   1:L PR[91] R[100]mm/sec CNT100;
   1:  PR[GP1:91,1] = PR[GP1:90,1] + -46.365;
   1:  PR[GP1:91,2] = PR[GP1:90,2] + -31.306;
   1:L PR[91] R[100]mm/sec CNT100;
   1:  PR[GP1:91,1] = PR[GP1:90,1] + -43.823;
   1:  PR[GP1:91,2] = PR[GP1:90,2] + -32.890;
   1:L PR[91] R[100]mm/sec CNT100;
   1:  PR[GP1:91,1] = PR[GP1:90,1] + -41.333;
   1:  PR[GP1:91,2] = PR[GP1:90,2] + -33.889;
   1:L PR[91] R[100]mm/sec CNT100;
   1:  PR[GP1:91,1] = PR[GP1:90,1] + -32.971;
   1:  PR[GP1:91,2] = PR[GP1:90,2] + -36.840;
   1:L PR[91] R[100]mm/sec CNT100;
   1:  PR[GP1:91,1] = PR[GP1:90,1] + -30.718;
   1:  PR[GP1:91,2] = PR[GP1:90,2] + -37.326;
   1:L PR[91] R[100]mm/sec CNT100;
   1:  PR[GP1:91,1] = PR[GP1:90,1] + -28.669;
   1:  PR[GP1:91,2] = PR[GP1:90,2] + -37.405;
   1:L PR[91] R[100]mm/sec CNT100;
   1:  PR[GP1:91,1] = PR[GP1:90,1] + -18.411;
   1:  PR[GP1:91,2] = PR[GP1:90,2] + -37.437;
   1:L PR[91] R[100]mm/sec CNT100;
   1:  PR[GP1:91,1] = PR[GP1:90,1] + -16.830;
   1:  PR[GP1:91,2] = PR[GP1:90,2] + -37.231;
   1:L PR[91] R[100]mm/sec CNT100;
   1:  PR[GP1:91,1] = PR[GP1:90,1] + -15.463;
   1:  PR[GP1:91,2] = PR[GP1:90,2] + -36.795;
   1:L PR[91] R[100]mm/sec CNT100;
   1:  PR[GP1:91,1] = PR[GP1:90,1] + -4.794;
   1:  PR[GP1:91,2] = PR[GP1:90,2] + -33.088;
   1:L PR[91] R[100]mm/sec CNT100;
   1:  PR[GP1:91,1] = PR[GP1:90,1] + -3.959;
   1:  PR[GP1:91,2] = PR[GP1:90,2] + -32.651;
   1:L PR[91] R[100]mm/sec CNT100;
   1:  PR[GP1:91,1] = PR[GP1:90,1] + -2.575;
   1:  PR[GP1:91,2] = PR[GP1:90,2] + -31.645;
   1:L PR[91] R[100]mm/sec CNT100;
   1:  PR[GP1:91,1] = PR[GP1:90,1] + -0.246;
   1:  PR[GP1:91,2] = PR[GP1:90,2] + -31.552;
   1:L PR[91] R[100]mm/sec CNT100;
   1:  PR[GP1:91,1] = PR[GP1:90,1] + 1.907;
   1:  PR[GP1:91,2] = PR[GP1:90,2] + -31.093;
   1:L PR[91] R[100]mm/sec CNT100;
   1:  PR[GP1:91,1] = PR[GP1:90,1] + 2.367;
   1:  PR[GP1:91,2] = PR[GP1:90,2] + -31.464;
   1:L PR[91] R[100]mm/sec CNT100;
   1:  PR[GP1:91,1] = PR[GP1:90,1] + 2.888;
   1:  PR[GP1:91,2] = PR[GP1:90,2] + -31.723;
   1:L PR[91] R[100]mm/sec CNT100;
   1:  PR[GP1:91,1] = PR[GP1:90,1] + 4.168;
   1:  PR[GP1:91,2] = PR[GP1:90,2] + -32.653;
   1:L PR[91] R[100]mm/sec CNT100;
   1:  PR[GP1:91,1] = PR[GP1:90,1] + 4.991;
   1:  PR[GP1:91,2] = PR[GP1:90,2] + -33.083;
   1:L PR[91] R[100]mm/sec CNT100;
   1:  PR[GP1:91,1] = PR[GP1:90,1] + 6.059;
   1:  PR[GP1:91,2] = PR[GP1:90,2] + -33.426;
   1:L PR[91] R[100]mm/sec CNT100;
   1:  PR[GP1:91,1] = PR[GP1:90,1] + 17.047;
   1:  PR[GP1:91,2] = PR[GP1:90,2] + -37.230;
   1:L PR[91] R[100]mm/sec CNT100;
   1:  PR[GP1:91,1] = PR[GP1:90,1] + 18.609;
   1:  PR[GP1:91,2] = PR[GP1:90,2] + -37.435;
   1:L PR[91] R[100]mm/sec CNT100;
   1:  PR[GP1:91,1] = PR[GP1:90,1] + 20.489;
   1:  PR[GP1:91,2] = PR[GP1:90,2] + -37.372;
   1:L PR[91] R[100]mm/sec CNT100;
   1:  PR[GP1:91,1] = PR[GP1:90,1] + 30.926;
   1:  PR[GP1:91,2] = PR[GP1:90,2] + -37.326;
   1:L PR[91] R[100]mm/sec CNT100;
   1:  PR[GP1:91,1] = PR[GP1:90,1] + 33.154;
   1:  PR[GP1:91,2] = PR[GP1:90,2] + -36.847;
   1:L PR[91] R[100]mm/sec CNT100;
   1:  PR[GP1:91,1] = PR[GP1:90,1] + 35.646;
   1:  PR[GP1:91,2] = PR[GP1:90,2] + -35.865;
   1:L PR[91] R[100]mm/sec CNT100;
   1:  PR[GP1:91,1] = PR[GP1:90,1] + 44.032;
   1:  PR[GP1:91,2] = PR[GP1:90,2] + -32.893;
   1:L PR[91] R[100]mm/sec CNT100;
   1:  PR[GP1:91,1] = PR[GP1:90,1] + 46.535;
   1:  PR[GP1:91,2] = PR[GP1:90,2] + -31.341;
   1:L PR[91] R[100]mm/sec CNT100;
   1:  PR[GP1:91,1] = PR[GP1:90,1] + 48.999;
   1:  PR[GP1:91,2] = PR[GP1:90,2] + -29.159;
   1:L PR[91] R[100]mm/sec CNT100;
   1:  PR[GP1:91,1] = PR[GP1:90,1] + 54.738;
   1:  PR[GP1:91,2] = PR[GP1:90,2] + -24.513;
   1:L PR[91] R[100]mm/sec CNT100;
   1:  PR[GP1:91,1] = PR[GP1:90,1] + 56.858;
   1:  PR[GP1:91,2] = PR[GP1:90,2] + -21.761;
   1:L PR[91] R[100]mm/sec CNT100;
   1:  PR[GP1:91,1] = PR[GP1:90,1] + 58.644;
   1:  PR[GP1:91,2] = PR[GP1:90,2] + -18.336;
   1:L PR[91] R[100]mm/sec CNT100;
   1:  PR[GP1:91,1] = PR[GP1:90,1] + 61.851;
   1:  PR[GP1:91,2] = PR[GP1:90,2] + -12.992;
   1:L PR[91] R[100]mm/sec CNT100;
   1:  PR[GP1:91,1] = PR[GP1:90,1] + 62.889;
   1:  PR[GP1:91,2] = PR[GP1:90,2] + -9.519;
   1:L PR[91] R[100]mm/sec CNT100;
   1:  PR[GP1:91,1] = PR[GP1:90,1] + 63.252;
   1:  PR[GP1:91,2] = PR[GP1:90,2] + -5.632;
   1:L PR[91] R[100]mm/sec CNT100;
   1:  PR[GP1:91,1] = PR[GP1:90,1] + 64.281;
   1:  PR[GP1:91,2] = PR[GP1:90,2] + -0.045;
   1:L PR[91] R[100]mm/sec CNT100;
   1:  PR[GP1:91,1] = PR[GP1:90,1] + 63.927;
   1:  PR[GP1:91,2] = PR[GP1:90,2] + 3.792;
   1:L PR[91] R[100]mm/sec CNT100;
   1:  PR[GP1:91,1] = PR[GP1:90,1] + 62.897;
   1:  PR[GP1:91,2] = PR[GP1:90,2] + 9.347;
   1:L PR[91] R[100]mm/sec CNT100;
   1:  PR[GP1:91,1] = PR[GP1:90,1] + 61.846;
   1:  PR[GP1:91,2] = PR[GP1:90,2] + 12.865;
   1:L PR[91] R[100]mm/sec CNT100;
   1:  PR[GP1:91,1] = PR[GP1:90,1] + 60.137;
   1:  PR[GP1:91,2] = PR[GP1:90,2] + 16.178;
   1:L PR[91] R[100]mm/sec CNT100;
   1:  PR[GP1:91,1] = PR[GP1:90,1] + 56.873;
   1:  PR[GP1:91,2] = PR[GP1:90,2] + 21.599;
   1:L PR[91] R[100]mm/sec CNT100;
   1:  PR[GP1:91,1] = PR[GP1:90,1] + 54.732;
   1:  PR[GP1:91,2] = PR[GP1:90,2] + 24.378;
   1:L PR[91] R[100]mm/sec CNT100;
   1:  PR[GP1:91,1] = PR[GP1:90,1] + 52.362;
   1:  PR[GP1:91,2] = PR[GP1:90,2] + 26.497;
   1:L PR[91] R[100]mm/sec CNT100;
   1:  PR[GP1:91,1] = PR[GP1:90,1] + 46.553;
   1:  PR[GP1:91,2] = PR[GP1:90,2] + 31.186;
   1:L PR[91] R[100]mm/sec CNT100;
   1:  PR[GP1:91,1] = PR[GP1:90,1] + 44.028;
   1:  PR[GP1:91,2] = PR[GP1:90,2] + 32.752;
   1:L PR[91] R[100]mm/sec CNT100;
   1:  PR[GP1:91,1] = PR[GP1:90,1] + 41.535;
   1:  PR[GP1:91,2] = PR[GP1:90,2] + 33.747;
   1:L PR[91] R[100]mm/sec CNT100;
   1:  PR[GP1:91,1] = PR[GP1:90,1] + 33.176;
   1:  PR[GP1:91,2] = PR[GP1:90,2] + 36.698;
   1:L PR[91] R[100]mm/sec CNT100;
   1:  PR[GP1:91,1] = PR[GP1:90,1] + 30.927;
   1:  PR[GP1:91,2] = PR[GP1:90,2] + 37.182;
   1:L PR[91] R[100]mm/sec CNT100;
   1:  PR[GP1:91,1] = PR[GP1:90,1] + 28.888;
   1:  PR[GP1:91,2] = PR[GP1:90,2] + 37.259;
   1:L PR[91] R[100]mm/sec CNT100;
   1:  PR[GP1:91,1] = PR[GP1:90,1] + 18.635;
   1:  PR[GP1:91,2] = PR[GP1:90,2] + 37.295;
   1:L PR[91] R[100]mm/sec CNT100;
   1:  PR[GP1:91,1] = PR[GP1:90,1] + 17.056;
   1:  PR[GP1:91,2] = PR[GP1:90,2] + 37.088;
   1:L PR[91] R[100]mm/sec CNT100;
   1:  PR[GP1:91,1] = PR[GP1:90,1] + 15.687;
   1:  PR[GP1:91,2] = PR[GP1:90,2] + 36.652;
   1:L PR[91] R[100]mm/sec CNT100;
   1:  PR[GP1:91,1] = PR[GP1:90,1] + 5.015;
   1:  PR[GP1:91,2] = PR[GP1:90,2] + 32.952;
   1:L PR[91] R[100]mm/sec CNT100;
   1:  PR[GP1:91,1] = PR[GP1:90,1] + 4.175;
   1:  PR[GP1:91,2] = PR[GP1:90,2] + 32.514;
   1:L PR[91] R[100]mm/sec CNT100;
   1:  PR[GP1:91,1] = PR[GP1:90,1] + 3.190;
   1:  PR[GP1:91,2] = PR[GP1:90,2] + 31.818;
   1:L PR[91] R[100]mm/sec CNT100;
   1:  PR[GP1:91,1] = PR[GP1:90,1] + 3.196;
   1:  PR[GP1:91,2] = PR[GP1:90,2] + 31.710;
   1:L PR[91] R[100]mm/sec CNT100;
   1:  PR[GP1:91,1] = PR[GP1:90,1] + 1.880;
   1:  PR[GP1:91,2] = PR[GP1:90,2] + 30.978;
   1:L PR[91] R[100]mm/sec CNT100;
   1:  ! -- Layer/Ebene 107 -- !;
   1:  PR[91] = PR[90];
   1:  PR[GP1:91,1] = PR[GP1:90,1] + -1.357;
   1:  PR[GP1:91,2] = PR[GP1:90,2] + 31.489;
   1:  PR[GP1:91,3] = PR[GP1:90,3] + 65.575;
   1:L PR[91] R[100]mm/sec CNT100;
   1:  PR[GP1:91,1] = PR[GP1:90,1] + -2.590;
   1:  PR[GP1:91,2] = PR[GP1:90,2] + 31.776;
   1:L PR[91] R[100]mm/sec CNT100;
   1:  PR[GP1:91,1] = PR[GP1:90,1] + -3.756;
   1:  PR[GP1:91,2] = PR[GP1:90,2] + 32.599;
   1:L PR[91] R[100]mm/sec CNT100;
   1:  PR[GP1:91,1] = PR[GP1:90,1] + -4.464;
   1:  PR[GP1:91,2] = PR[GP1:90,2] + 32.970;
   1:L PR[91] R[100]mm/sec CNT100;
   1:  PR[GP1:91,1] = PR[GP1:90,1] + -5.379;
   1:  PR[GP1:91,2] = PR[GP1:90,2] + 33.264;
   1:L PR[91] R[100]mm/sec CNT100;
   1:  PR[GP1:91,1] = PR[GP1:90,1] + -16.656;
   1:  PR[GP1:91,2] = PR[GP1:90,2] + 37.163;
   1:L PR[91] R[100]mm/sec CNT100;
   1:  PR[GP1:91,1] = PR[GP1:90,1] + -18.068;
   1:  PR[GP1:91,2] = PR[GP1:90,2] + 37.347;
   1:L PR[91] R[100]mm/sec CNT100;
   1:  PR[GP1:91,1] = PR[GP1:90,1] + -19.782;
   1:  PR[GP1:91,2] = PR[GP1:90,2] + 37.288;
   1:L PR[91] R[100]mm/sec CNT100;
   1:  PR[GP1:91,1] = PR[GP1:90,1] + -30.552;
   1:  PR[GP1:91,2] = PR[GP1:90,2] + 37.234;
   1:L PR[91] R[100]mm/sec CNT100;
   1:  PR[GP1:91,1] = PR[GP1:90,1] + -32.626;
   1:  PR[GP1:91,2] = PR[GP1:90,2] + 36.787;
   1:L PR[91] R[100]mm/sec CNT100;
   1:  PR[GP1:91,1] = PR[GP1:90,1] + -34.945;
   1:  PR[GP1:91,2] = PR[GP1:90,2] + 35.869;
   1:L PR[91] R[100]mm/sec CNT100;
   1:  PR[GP1:91,1] = PR[GP1:90,1] + -43.657;
   1:  PR[GP1:91,2] = PR[GP1:90,2] + 32.775;
   1:L PR[91] R[100]mm/sec CNT100;
   1:  PR[GP1:91,1] = PR[GP1:90,1] + -46.035;
   1:  PR[GP1:91,2] = PR[GP1:90,2] + 31.294;
   1:L PR[91] R[100]mm/sec CNT100;
   1:  PR[GP1:91,1] = PR[GP1:90,1] + -48.377;
   1:  PR[GP1:91,2] = PR[GP1:90,2] + 29.214;
   1:L PR[91] R[100]mm/sec CNT100;
   1:  PR[GP1:91,1] = PR[GP1:90,1] + -54.388;
   1:  PR[GP1:91,2] = PR[GP1:90,2] + 24.350;
   1:L PR[91] R[100]mm/sec CNT100;
   1:  PR[GP1:91,1] = PR[GP1:90,1] + -56.385;
   1:  PR[GP1:91,2] = PR[GP1:90,2] + 21.751;
   1:L PR[91] R[100]mm/sec CNT100;
   1:  PR[GP1:91,1] = PR[GP1:90,1] + -58.081;
   1:  PR[GP1:91,2] = PR[GP1:90,2] + 18.459;
   1:L PR[91] R[100]mm/sec CNT100;
   1:  PR[GP1:91,1] = PR[GP1:90,1] + -61.467;
   1:  PR[GP1:91,2] = PR[GP1:90,2] + 12.803;
   1:L PR[91] R[100]mm/sec CNT100;
   1:  PR[GP1:91,1] = PR[GP1:90,1] + -62.460;
   1:  PR[GP1:91,2] = PR[GP1:90,2] + 9.434;
   1:L PR[91] R[100]mm/sec CNT100;
   1:  PR[GP1:91,1] = PR[GP1:90,1] + -62.791;
   1:  PR[GP1:91,2] = PR[GP1:90,2] + 5.814;
   1:L PR[91] R[100]mm/sec CNT100;
   1:  PR[GP1:91,1] = PR[GP1:90,1] + -63.881;
   1:  PR[GP1:91,2] = PR[GP1:90,2] + -0.100;
   1:L PR[91] R[100]mm/sec CNT100;
   1:  PR[GP1:91,1] = PR[GP1:90,1] + -63.558;
   1:  PR[GP1:91,2] = PR[GP1:90,2] + -3.675;
   1:L PR[91] R[100]mm/sec CNT100;
   1:  PR[GP1:91,1] = PR[GP1:90,1] + -62.467;
   1:  PR[GP1:91,2] = PR[GP1:90,2] + -9.553;
   1:L PR[91] R[100]mm/sec CNT100;
   1:  PR[GP1:91,1] = PR[GP1:90,1] + -61.460;
   1:  PR[GP1:91,2] = PR[GP1:90,2] + -12.969;
   1:L PR[91] R[100]mm/sec CNT100;
   1:  PR[GP1:91,1] = PR[GP1:90,1] + -59.830;
   1:  PR[GP1:91,2] = PR[GP1:90,2] + -16.165;
   1:L PR[91] R[100]mm/sec CNT100;
   1:  PR[GP1:91,1] = PR[GP1:90,1] + -56.394;
   1:  PR[GP1:91,2] = PR[GP1:90,2] + -21.883;
   1:L PR[91] R[100]mm/sec CNT100;
   1:  PR[GP1:91,1] = PR[GP1:90,1] + -54.376;
   1:  PR[GP1:91,2] = PR[GP1:90,2] + -24.509;
   1:L PR[91] R[100]mm/sec CNT100;
   1:  PR[GP1:91,1] = PR[GP1:90,1] + -52.106;
   1:  PR[GP1:91,2] = PR[GP1:90,2] + -26.545;
   1:L PR[91] R[100]mm/sec CNT100;
   1:  PR[GP1:91,1] = PR[GP1:90,1] + -46.040;
   1:  PR[GP1:91,2] = PR[GP1:90,2] + -31.434;
   1:L PR[91] R[100]mm/sec CNT100;
   1:  PR[GP1:91,1] = PR[GP1:90,1] + -43.639;
   1:  PR[GP1:91,2] = PR[GP1:90,2] + -32.930;
   1:L PR[91] R[100]mm/sec CNT100;
   1:  PR[GP1:91,1] = PR[GP1:90,1] + -41.287;
   1:  PR[GP1:91,2] = PR[GP1:90,2] + -33.874;
   1:L PR[91] R[100]mm/sec CNT100;
   1:  PR[GP1:91,1] = PR[GP1:90,1] + -32.625;
   1:  PR[GP1:91,2] = PR[GP1:90,2] + -36.931;
   1:L PR[91] R[100]mm/sec CNT100;
   1:  PR[GP1:91,1] = PR[GP1:90,1] + -30.530;
   1:  PR[GP1:91,2] = PR[GP1:90,2] + -37.383;
   1:L PR[91] R[100]mm/sec CNT100;
   1:  PR[GP1:91,1] = PR[GP1:90,1] + -28.623;
   1:  PR[GP1:91,2] = PR[GP1:90,2] + -37.456;
   1:L PR[91] R[100]mm/sec CNT100;
   1:  PR[GP1:91,1] = PR[GP1:90,1] + -18.059;
   1:  PR[GP1:91,2] = PR[GP1:90,2] + -37.489;
   1:L PR[91] R[100]mm/sec CNT100;
   1:  PR[GP1:91,1] = PR[GP1:90,1] + -16.631;
   1:  PR[GP1:91,2] = PR[GP1:90,2] + -37.303;
   1:L PR[91] R[100]mm/sec CNT100;
   1:  PR[GP1:91,1] = PR[GP1:90,1] + -15.394;
   1:  PR[GP1:91,2] = PR[GP1:90,2] + -36.909;
   1:L PR[91] R[100]mm/sec CNT100;
   1:  PR[GP1:91,1] = PR[GP1:90,1] + -4.452;
   1:  PR[GP1:91,2] = PR[GP1:90,2] + -33.107;
   1:L PR[91] R[100]mm/sec CNT100;
   1:  PR[GP1:91,1] = PR[GP1:90,1] + -3.748;
   1:  PR[GP1:91,2] = PR[GP1:90,2] + -32.739;
   1:L PR[91] R[100]mm/sec CNT100;
   1:  PR[GP1:91,1] = PR[GP1:90,1] + -2.547;
   1:  PR[GP1:91,2] = PR[GP1:90,2] + -31.865;
   1:L PR[91] R[100]mm/sec CNT100;
   1:  PR[GP1:91,1] = PR[GP1:90,1] + -0.081;
   1:  PR[GP1:91,2] = PR[GP1:90,2] + -31.767;
   1:L PR[91] R[100]mm/sec CNT100;
   1:  PR[GP1:91,1] = PR[GP1:90,1] + 1.937;
   1:  PR[GP1:91,2] = PR[GP1:90,2] + -31.336;
   1:L PR[91] R[100]mm/sec CNT100;
   1:  PR[GP1:91,1] = PR[GP1:90,1] + 2.416;
   1:  PR[GP1:91,2] = PR[GP1:90,2] + -31.722;
   1:L PR[91] R[100]mm/sec CNT100;
   1:  PR[GP1:91,1] = PR[GP1:90,1] + 2.859;
   1:  PR[GP1:91,2] = PR[GP1:90,2] + -31.943;
   1:L PR[91] R[100]mm/sec CNT100;
   1:  PR[GP1:91,1] = PR[GP1:90,1] + 3.957;
   1:  PR[GP1:91,2] = PR[GP1:90,2] + -32.740;
   1:L PR[91] R[100]mm/sec CNT100;
   1:  PR[GP1:91,1] = PR[GP1:90,1] + 4.649;
   1:  PR[GP1:91,2] = PR[GP1:90,2] + -33.101;
   1:L PR[91] R[100]mm/sec CNT100;
   1:  PR[GP1:91,1] = PR[GP1:90,1] + 5.557;
   1:  PR[GP1:91,2] = PR[GP1:90,2] + -33.393;
   1:L PR[91] R[100]mm/sec CNT100;
   1:  PR[GP1:91,1] = PR[GP1:90,1] + 16.848;
   1:  PR[GP1:91,2] = PR[GP1:90,2] + -37.302;
   1:L PR[91] R[100]mm/sec CNT100;
   1:  PR[GP1:91,1] = PR[GP1:90,1] + 18.257;
   1:  PR[GP1:91,2] = PR[GP1:90,2] + -37.487;
   1:L PR[91] R[100]mm/sec CNT100;
   1:  PR[GP1:91,1] = PR[GP1:90,1] + 19.962;
   1:  PR[GP1:91,2] = PR[GP1:90,2] + -37.430;
   1:L PR[91] R[100]mm/sec CNT100;
   1:  PR[GP1:91,1] = PR[GP1:90,1] + 30.738;
   1:  PR[GP1:91,2] = PR[GP1:90,2] + -37.383;
   1:L PR[91] R[100]mm/sec CNT100;
   1:  PR[GP1:91,1] = PR[GP1:90,1] + 32.809;
   1:  PR[GP1:91,2] = PR[GP1:90,2] + -36.937;
   1:L PR[91] R[100]mm/sec CNT100;
   1:  PR[GP1:91,1] = PR[GP1:90,1] + 35.130;
   1:  PR[GP1:91,2] = PR[GP1:90,2] + -36.023;
   1:L PR[91] R[100]mm/sec CNT100;
   1:  PR[GP1:91,1] = PR[GP1:90,1] + 43.849;
   1:  PR[GP1:91,2] = PR[GP1:90,2] + -32.933;
   1:L PR[91] R[100]mm/sec CNT100;
   1:  PR[GP1:91,1] = PR[GP1:90,1] + 46.211;
   1:  PR[GP1:91,2] = PR[GP1:90,2] + -31.468;
   1:L PR[91] R[100]mm/sec CNT100;
   1:  PR[GP1:91,1] = PR[GP1:90,1] + 48.541;
   1:  PR[GP1:91,2] = PR[GP1:90,2] + -29.406;
   1:L PR[91] R[100]mm/sec CNT100;
   1:  PR[GP1:91,1] = PR[GP1:90,1] + 54.557;
   1:  PR[GP1:91,2] = PR[GP1:90,2] + -24.536;
   1:L PR[91] R[100]mm/sec CNT100;
   1:  PR[GP1:91,1] = PR[GP1:90,1] + 56.575;
   1:  PR[GP1:91,2] = PR[GP1:90,2] + -21.916;
   1:L PR[91] R[100]mm/sec CNT100;
   1:  PR[GP1:91,1] = PR[GP1:90,1] + 58.276;
   1:  PR[GP1:91,2] = PR[GP1:90,2] + -18.651;
   1:L PR[91] R[100]mm/sec CNT100;
   1:  PR[GP1:91,1] = PR[GP1:90,1] + 61.665;
   1:  PR[GP1:91,2] = PR[GP1:90,2] + -13.006;
   1:L PR[91] R[100]mm/sec CNT100;
   1:  PR[GP1:91,1] = PR[GP1:90,1] + 62.656;
   1:  PR[GP1:91,2] = PR[GP1:90,2] + -9.687;
   1:L PR[91] R[100]mm/sec CNT100;
   1:  PR[GP1:91,1] = PR[GP1:90,1] + 63.004;
   1:  PR[GP1:91,2] = PR[GP1:90,2] + -5.967;
   1:L PR[91] R[100]mm/sec CNT100;
   1:  PR[GP1:91,1] = PR[GP1:90,1] + 64.095;
   1:  PR[GP1:91,2] = PR[GP1:90,2] + -0.045;
   1:L PR[91] R[100]mm/sec CNT100;
   1:  PR[GP1:91,1] = PR[GP1:90,1] + 63.755;
   1:  PR[GP1:91,2] = PR[GP1:90,2] + 3.631;
   1:L PR[91] R[100]mm/sec CNT100;
   1:  PR[GP1:91,1] = PR[GP1:90,1] + 62.665;
   1:  PR[GP1:91,2] = PR[GP1:90,2] + 9.515;
   1:L PR[91] R[100]mm/sec CNT100;
   1:  PR[GP1:91,1] = PR[GP1:90,1] + 61.660;
   1:  PR[GP1:91,2] = PR[GP1:90,2] + 12.879;
   1:L PR[91] R[100]mm/sec CNT100;
   1:  PR[GP1:91,1] = PR[GP1:90,1] + 60.025;
   1:  PR[GP1:91,2] = PR[GP1:90,2] + 16.047;
   1:L PR[91] R[100]mm/sec CNT100;
   1:  PR[GP1:91,1] = PR[GP1:90,1] + 56.589;
   1:  PR[GP1:91,2] = PR[GP1:90,2] + 21.754;
   1:L PR[91] R[100]mm/sec CNT100;
   1:  PR[GP1:91,1] = PR[GP1:90,1] + 54.551;
   1:  PR[GP1:91,2] = PR[GP1:90,2] + 24.400;
   1:L PR[91] R[100]mm/sec CNT100;
   1:  PR[GP1:91,1] = PR[GP1:90,1] + 52.293;
   1:  PR[GP1:91,2] = PR[GP1:90,2] + 26.419;
   1:L PR[91] R[100]mm/sec CNT100;
   1:  PR[GP1:91,1] = PR[GP1:90,1] + 46.230;
   1:  PR[GP1:91,2] = PR[GP1:90,2] + 31.313;
   1:L PR[91] R[100]mm/sec CNT100;
   1:  PR[GP1:91,1] = PR[GP1:90,1] + 43.845;
   1:  PR[GP1:91,2] = PR[GP1:90,2] + 32.791;
   1:L PR[91] R[100]mm/sec CNT100;
   1:  PR[GP1:91,1] = PR[GP1:90,1] + 41.490;
   1:  PR[GP1:91,2] = PR[GP1:90,2] + 33.732;
   1:L PR[91] R[100]mm/sec CNT100;
   1:  PR[GP1:91,1] = PR[GP1:90,1] + 32.832;
   1:  PR[GP1:91,2] = PR[GP1:90,2] + 36.789;
   1:L PR[91] R[100]mm/sec CNT100;
   1:  PR[GP1:91,1] = PR[GP1:90,1] + 30.741;
   1:  PR[GP1:91,2] = PR[GP1:90,2] + 37.239;
   1:L PR[91] R[100]mm/sec CNT100;
   1:  PR[GP1:91,1] = PR[GP1:90,1] + 28.843;
   1:  PR[GP1:91,2] = PR[GP1:90,2] + 37.310;
   1:L PR[91] R[100]mm/sec CNT100;
   1:  PR[GP1:91,1] = PR[GP1:90,1] + 18.284;
   1:  PR[GP1:91,2] = PR[GP1:90,2] + 37.347;
   1:L PR[91] R[100]mm/sec CNT100;
   1:  PR[GP1:91,1] = PR[GP1:90,1] + 16.857;
   1:  PR[GP1:91,2] = PR[GP1:90,2] + 37.160;
   1:L PR[91] R[100]mm/sec CNT100;
   1:  PR[GP1:91,1] = PR[GP1:90,1] + 15.618;
   1:  PR[GP1:91,2] = PR[GP1:90,2] + 36.766;
   1:L PR[91] R[100]mm/sec CNT100;
   1:  PR[GP1:91,1] = PR[GP1:90,1] + 4.674;
   1:  PR[GP1:91,2] = PR[GP1:90,2] + 32.971;
   1:L PR[91] R[100]mm/sec CNT100;
   1:  PR[GP1:91,1] = PR[GP1:90,1] + 3.964;
   1:  PR[GP1:91,2] = PR[GP1:90,2] + 32.601;
   1:L PR[91] R[100]mm/sec CNT100;
   1:  PR[GP1:91,1] = PR[GP1:90,1] + 3.162;
   1:  PR[GP1:91,2] = PR[GP1:90,2] + 32.035;
   1:L PR[91] R[100]mm/sec CNT100;
   1:  PR[GP1:91,1] = PR[GP1:90,1] + 3.168;
   1:  PR[GP1:91,2] = PR[GP1:90,2] + 31.921;
   1:L PR[91] R[100]mm/sec CNT100;
   1:  PR[GP1:91,1] = PR[GP1:90,1] + 1.910;
   1:  PR[GP1:91,2] = PR[GP1:90,2] + 31.221;
   1:L PR[91] R[100]mm/sec CNT100;
   1:  ! -- Layer/Ebene 108 -- !;
   1:  PR[91] = PR[90];
   1:  PR[GP1:91,1] = PR[GP1:90,1] + -1.508;
   1:  PR[GP1:91,2] = PR[GP1:90,2] + 31.747;
   1:  PR[GP1:91,3] = PR[GP1:90,3] + 66.185;
   1:L PR[91] R[100]mm/sec CNT100;
   1:  PR[GP1:91,1] = PR[GP1:90,1] + -2.562;
   1:  PR[GP1:91,2] = PR[GP1:90,2] + 31.993;
   1:L PR[91] R[100]mm/sec CNT100;
   1:  PR[GP1:91,1] = PR[GP1:90,1] + -3.545;
   1:  PR[GP1:91,2] = PR[GP1:90,2] + 32.687;
   1:L PR[91] R[100]mm/sec CNT100;
   1:  PR[GP1:91,1] = PR[GP1:90,1] + -4.122;
   1:  PR[GP1:91,2] = PR[GP1:90,2] + 32.989;
   1:L PR[91] R[100]mm/sec CNT100;
   1:  PR[GP1:91,1] = PR[GP1:90,1] + -4.879;
   1:  PR[GP1:91,2] = PR[GP1:90,2] + 33.232;
   1:L PR[91] R[100]mm/sec CNT100;
   1:  PR[GP1:91,1] = PR[GP1:90,1] + -16.457;
   1:  PR[GP1:91,2] = PR[GP1:90,2] + 37.235;
   1:L PR[91] R[100]mm/sec CNT100;
   1:  PR[GP1:91,1] = PR[GP1:90,1] + -17.717;
   1:  PR[GP1:91,2] = PR[GP1:90,2] + 37.399;
   1:L PR[91] R[100]mm/sec CNT100;
   1:  PR[GP1:91,1] = PR[GP1:90,1] + -19.253;
   1:  PR[GP1:91,2] = PR[GP1:90,2] + 37.346;
   1:L PR[91] R[100]mm/sec CNT100;
   1:  PR[GP1:91,1] = PR[GP1:90,1] + -30.365;
   1:  PR[GP1:91,2] = PR[GP1:90,2] + 37.291;
   1:L PR[91] R[100]mm/sec CNT100;
   1:  PR[GP1:91,1] = PR[GP1:90,1] + -32.281;
   1:  PR[GP1:91,2] = PR[GP1:90,2] + 36.877;
   1:L PR[91] R[100]mm/sec CNT100;
   1:  PR[GP1:91,1] = PR[GP1:90,1] + -34.429;
   1:  PR[GP1:91,2] = PR[GP1:90,2] + 36.027;
   1:L PR[91] R[100]mm/sec CNT100;
   1:  PR[GP1:91,1] = PR[GP1:90,1] + -43.474;
   1:  PR[GP1:91,2] = PR[GP1:90,2] + 32.815;
   1:L PR[91] R[100]mm/sec CNT100;
   1:  PR[GP1:91,1] = PR[GP1:90,1] + -45.710;
   1:  PR[GP1:91,2] = PR[GP1:90,2] + 31.422;
   1:L PR[91] R[100]mm/sec CNT100;
   1:  PR[GP1:91,1] = PR[GP1:90,1] + -47.917;
   1:  PR[GP1:91,2] = PR[GP1:90,2] + 29.462;
   1:L PR[91] R[100]mm/sec CNT100;
   1:  PR[GP1:91,1] = PR[GP1:90,1] + -54.205;
   1:  PR[GP1:91,2] = PR[GP1:90,2] + 24.374;
   1:L PR[91] R[100]mm/sec CNT100;
   1:  PR[GP1:91,1] = PR[GP1:90,1] + -56.100;
   1:  PR[GP1:91,2] = PR[GP1:90,2] + 21.907;
   1:L PR[91] R[100]mm/sec CNT100;
   1:  PR[GP1:91,1] = PR[GP1:90,1] + -57.713;
   1:  PR[GP1:91,2] = PR[GP1:90,2] + 18.777;
   1:L PR[91] R[100]mm/sec CNT100;
   1:  PR[GP1:91,1] = PR[GP1:90,1] + -61.280;
   1:  PR[GP1:91,2] = PR[GP1:90,2] + 12.819;
   1:L PR[91] R[100]mm/sec CNT100;
   1:  PR[GP1:91,1] = PR[GP1:90,1] + -62.227;
   1:  PR[GP1:91,2] = PR[GP1:90,2] + 9.605;
   1:L PR[91] R[100]mm/sec CNT100;
   1:  PR[GP1:91,1] = PR[GP1:90,1] + -62.543;
   1:  PR[GP1:91,2] = PR[GP1:90,2] + 6.148;
   1:L PR[91] R[100]mm/sec CNT100;
   1:  PR[GP1:91,1] = PR[GP1:90,1] + -63.695;
   1:  PR[GP1:91,2] = PR[GP1:90,2] + -0.100;
   1:L PR[91] R[100]mm/sec CNT100;
   1:  PR[GP1:91,1] = PR[GP1:90,1] + -63.386;
   1:  PR[GP1:91,2] = PR[GP1:90,2] + -3.518;
   1:L PR[91] R[100]mm/sec CNT100;
   1:  PR[GP1:91,1] = PR[GP1:90,1] + -62.234;
   1:  PR[GP1:91,2] = PR[GP1:90,2] + -9.725;
   1:L PR[91] R[100]mm/sec CNT100;
   1:  PR[GP1:91,1] = PR[GP1:90,1] + -61.273;
   1:  PR[GP1:91,2] = PR[GP1:90,2] + -12.985;
   1:L PR[91] R[100]mm/sec CNT100;
   1:  PR[GP1:91,1] = PR[GP1:90,1] + -59.717;
   1:  PR[GP1:91,2] = PR[GP1:90,2] + -16.035;
   1:L PR[91] R[100]mm/sec CNT100;
   1:  PR[GP1:91,1] = PR[GP1:90,1] + -56.109;
   1:  PR[GP1:91,2] = PR[GP1:90,2] + -22.039;
   1:L PR[91] R[100]mm/sec CNT100;
   1:  PR[GP1:91,1] = PR[GP1:90,1] + -54.192;
   1:  PR[GP1:91,2] = PR[GP1:90,2] + -24.534;
   1:L PR[91] R[100]mm/sec CNT100;
   1:  PR[GP1:91,1] = PR[GP1:90,1] + -52.036;
   1:  PR[GP1:91,2] = PR[GP1:90,2] + -26.468;
   1:L PR[91] R[100]mm/sec CNT100;
   1:  PR[GP1:91,1] = PR[GP1:90,1] + -45.715;
   1:  PR[GP1:91,2] = PR[GP1:90,2] + -31.563;
   1:L PR[91] R[100]mm/sec CNT100;
   1:  PR[GP1:91,1] = PR[GP1:90,1] + -43.456;
   1:  PR[GP1:91,2] = PR[GP1:90,2] + -32.970;
   1:L PR[91] R[100]mm/sec CNT100;
   1:  PR[GP1:91,1] = PR[GP1:90,1] + -41.242;
   1:  PR[GP1:91,2] = PR[GP1:90,2] + -33.859;
   1:L PR[91] R[100]mm/sec CNT100;
   1:  PR[GP1:91,1] = PR[GP1:90,1] + -32.279;
   1:  PR[GP1:91,2] = PR[GP1:90,2] + -37.021;
   1:L PR[91] R[100]mm/sec CNT100;
   1:  PR[GP1:91,1] = PR[GP1:90,1] + -30.342;
   1:  PR[GP1:91,2] = PR[GP1:90,2] + -37.439;
   1:L PR[91] R[100]mm/sec CNT100;
   1:  PR[GP1:91,1] = PR[GP1:90,1] + -28.577;
   1:  PR[GP1:91,2] = PR[GP1:90,2] + -37.507;
   1:L PR[91] R[100]mm/sec CNT100;
   1:  PR[GP1:91,1] = PR[GP1:90,1] + -17.707;
   1:  PR[GP1:91,2] = PR[GP1:90,2] + -37.542;
   1:L PR[91] R[100]mm/sec CNT100;
   1:  PR[GP1:91,1] = PR[GP1:90,1] + -16.432;
   1:  PR[GP1:91,2] = PR[GP1:90,2] + -37.375;
   1:L PR[91] R[100]mm/sec CNT100;
   1:  PR[GP1:91,1] = PR[GP1:90,1] + -15.326;
   1:  PR[GP1:91,2] = PR[GP1:90,2] + -37.023;
   1:L PR[91] R[100]mm/sec CNT100;
   1:  PR[GP1:91,1] = PR[GP1:90,1] + -4.110;
   1:  PR[GP1:91,2] = PR[GP1:90,2] + -33.125;
   1:L PR[91] R[100]mm/sec CNT100;
   1:  PR[GP1:91,1] = PR[GP1:90,1] + -3.538;
   1:  PR[GP1:91,2] = PR[GP1:90,2] + -32.826;
   1:L PR[91] R[100]mm/sec CNT100;
   1:  PR[GP1:91,1] = PR[GP1:90,1] + -2.519;
   1:  PR[GP1:91,2] = PR[GP1:90,2] + -32.086;
   1:L PR[91] R[100]mm/sec CNT100;
   1:  PR[GP1:91,1] = PR[GP1:90,1] + 0.085;
   1:  PR[GP1:91,2] = PR[GP1:90,2] + -31.982;
   1:L PR[91] R[100]mm/sec CNT100;
   1:  PR[GP1:91,1] = PR[GP1:90,1] + 1.967;
   1:  PR[GP1:91,2] = PR[GP1:90,2] + -31.580;
   1:L PR[91] R[100]mm/sec CNT100;
   1:  PR[GP1:91,1] = PR[GP1:90,1] + 2.464;
   1:  PR[GP1:91,2] = PR[GP1:90,2] + -31.980;
   1:L PR[91] R[100]mm/sec CNT100;
   1:  PR[GP1:91,1] = PR[GP1:90,1] + 2.831;
   1:  PR[GP1:91,2] = PR[GP1:90,2] + -32.163;
   1:L PR[91] R[100]mm/sec CNT100;
   1:  PR[GP1:91,1] = PR[GP1:90,1] + 3.745;
   1:  PR[GP1:91,2] = PR[GP1:90,2] + -32.827;
   1:L PR[91] R[100]mm/sec CNT100;
   1:  PR[GP1:91,1] = PR[GP1:90,1] + 4.307;
   1:  PR[GP1:91,2] = PR[GP1:90,2] + -33.120;
   1:L PR[91] R[100]mm/sec CNT100;
   1:  PR[GP1:91,1] = PR[GP1:90,1] + 5.055;
   1:  PR[GP1:91,2] = PR[GP1:90,2] + -33.360;
   1:L PR[91] R[100]mm/sec CNT100;
   1:  PR[GP1:91,1] = PR[GP1:90,1] + 16.649;
   1:  PR[GP1:91,2] = PR[GP1:90,2] + -37.374;
   1:L PR[91] R[100]mm/sec CNT100;
   1:  PR[GP1:91,1] = PR[GP1:90,1] + 17.906;
   1:  PR[GP1:91,2] = PR[GP1:90,2] + -37.540;
   1:L PR[91] R[100]mm/sec CNT100;
   1:  PR[GP1:91,1] = PR[GP1:90,1] + 19.434;
   1:  PR[GP1:91,2] = PR[GP1:90,2] + -37.488;
   1:L PR[91] R[100]mm/sec CNT100;
   1:  PR[GP1:91,1] = PR[GP1:90,1] + 30.551;
   1:  PR[GP1:91,2] = PR[GP1:90,2] + -37.439;
   1:L PR[91] R[100]mm/sec CNT100;
   1:  PR[GP1:91,1] = PR[GP1:90,1] + 32.464;
   1:  PR[GP1:91,2] = PR[GP1:90,2] + -37.028;
   1:L PR[91] R[100]mm/sec CNT100;
   1:  PR[GP1:91,1] = PR[GP1:90,1] + 34.615;
   1:  PR[GP1:91,2] = PR[GP1:90,2] + -36.180;
   1:L PR[91] R[100]mm/sec CNT100;
   1:  PR[GP1:91,1] = PR[GP1:90,1] + 43.666;
   1:  PR[GP1:91,2] = PR[GP1:90,2] + -32.973;
   1:L PR[91] R[100]mm/sec CNT100;
   1:  PR[GP1:91,1] = PR[GP1:90,1] + 45.888;
   1:  PR[GP1:91,2] = PR[GP1:90,2] + -31.595;
   1:L PR[91] R[100]mm/sec CNT100;
   1:  PR[GP1:91,1] = PR[GP1:90,1] + 48.082;
   1:  PR[GP1:91,2] = PR[GP1:90,2] + -29.652;
   1:L PR[91] R[100]mm/sec CNT100;
   1:  PR[GP1:91,1] = PR[GP1:90,1] + 54.375;
   1:  PR[GP1:91,2] = PR[GP1:90,2] + -24.558;
   1:L PR[91] R[100]mm/sec CNT100;
   1:  PR[GP1:91,1] = PR[GP1:90,1] + 56.291;
   1:  PR[GP1:91,2] = PR[GP1:90,2] + -22.071;
   1:L PR[91] R[100]mm/sec CNT100;
   1:  PR[GP1:91,1] = PR[GP1:90,1] + 57.908;
   1:  PR[GP1:91,2] = PR[GP1:90,2] + -18.967;
   1:L PR[91] R[100]mm/sec CNT100;
   1:  PR[GP1:91,1] = PR[GP1:90,1] + 61.478;
   1:  PR[GP1:91,2] = PR[GP1:90,2] + -13.020;
   1:L PR[91] R[100]mm/sec CNT100;
   1:  PR[GP1:91,1] = PR[GP1:90,1] + 62.424;
   1:  PR[GP1:91,2] = PR[GP1:90,2] + -9.854;
   1:L PR[91] R[100]mm/sec CNT100;
   1:  PR[GP1:91,1] = PR[GP1:90,1] + 62.756;
   1:  PR[GP1:91,2] = PR[GP1:90,2] + -6.302;
   1:L PR[91] R[100]mm/sec CNT100;
   1:  PR[GP1:91,1] = PR[GP1:90,1] + 63.908;
   1:  PR[GP1:91,2] = PR[GP1:90,2] + -0.045;
   1:L PR[91] R[100]mm/sec CNT100;
   1:  PR[GP1:91,1] = PR[GP1:90,1] + 63.584;
   1:  PR[GP1:91,2] = PR[GP1:90,2] + 3.470;
   1:L PR[91] R[100]mm/sec CNT100;
   1:  PR[GP1:91,1] = PR[GP1:90,1] + 62.433;
   1:  PR[GP1:91,2] = PR[GP1:90,2] + 9.682;
   1:L PR[91] R[100]mm/sec CNT100;
   1:  PR[GP1:91,1] = PR[GP1:90,1] + 61.474;
   1:  PR[GP1:91,2] = PR[GP1:90,2] + 12.892;
   1:L PR[91] R[100]mm/sec CNT100;
   1:  PR[GP1:91,1] = PR[GP1:90,1] + 59.913;
   1:  PR[GP1:91,2] = PR[GP1:90,2] + 15.917;
   1:L PR[91] R[100]mm/sec CNT100;
   1:  PR[GP1:91,1] = PR[GP1:90,1] + 56.305;
   1:  PR[GP1:91,2] = PR[GP1:90,2] + 21.909;
   1:L PR[91] R[100]mm/sec CNT100;
   1:  PR[GP1:91,1] = PR[GP1:90,1] + 54.369;
   1:  PR[GP1:91,2] = PR[GP1:90,2] + 24.422;
   1:L PR[91] R[100]mm/sec CNT100;
   1:  PR[GP1:91,1] = PR[GP1:90,1] + 52.225;
   1:  PR[GP1:91,2] = PR[GP1:90,2] + 26.340;
   1:L PR[91] R[100]mm/sec CNT100;
   1:  PR[GP1:91,1] = PR[GP1:90,1] + 45.907;
   1:  PR[GP1:91,2] = PR[GP1:90,2] + 31.440;
   1:L PR[91] R[100]mm/sec CNT100;
   1:  PR[GP1:91,1] = PR[GP1:90,1] + 43.663;
   1:  PR[GP1:91,2] = PR[GP1:90,2] + 32.831;
   1:L PR[91] R[100]mm/sec CNT100;
   1:  PR[GP1:91,1] = PR[GP1:90,1] + 41.445;
   1:  PR[GP1:91,2] = PR[GP1:90,2] + 33.716;
   1:L PR[91] R[100]mm/sec CNT100;
   1:  PR[GP1:91,1] = PR[GP1:90,1] + 32.487;
   1:  PR[GP1:91,2] = PR[GP1:90,2] + 36.879;
   1:L PR[91] R[100]mm/sec CNT100;
   1:  PR[GP1:91,1] = PR[GP1:90,1] + 30.554;
   1:  PR[GP1:91,2] = PR[GP1:90,2] + 37.295;
   1:L PR[91] R[100]mm/sec CNT100;
   1:  PR[GP1:91,1] = PR[GP1:90,1] + 28.798;
   1:  PR[GP1:91,2] = PR[GP1:90,2] + 37.362;
   1:L PR[91] R[100]mm/sec CNT100;
   1:  PR[GP1:91,1] = PR[GP1:90,1] + 17.933;
   1:  PR[GP1:91,2] = PR[GP1:90,2] + 37.400;
   1:L PR[91] R[100]mm/sec CNT100;
   1:  PR[GP1:91,1] = PR[GP1:90,1] + 16.659;
   1:  PR[GP1:91,2] = PR[GP1:90,2] + 37.232;
   1:L PR[91] R[100]mm/sec CNT100;
   1:  PR[GP1:91,1] = PR[GP1:90,1] + 15.551;
   1:  PR[GP1:91,2] = PR[GP1:90,2] + 36.880;
   1:L PR[91] R[100]mm/sec CNT100;
   1:  PR[GP1:91,1] = PR[GP1:90,1] + 4.332;
   1:  PR[GP1:91,2] = PR[GP1:90,2] + 32.990;
   1:L PR[91] R[100]mm/sec CNT100;
   1:  PR[GP1:91,1] = PR[GP1:90,1] + 3.752;
   1:  PR[GP1:91,2] = PR[GP1:90,2] + 32.688;
   1:L PR[91] R[100]mm/sec CNT100;
   1:  PR[GP1:91,1] = PR[GP1:90,1] + 3.134;
   1:  PR[GP1:91,2] = PR[GP1:90,2] + 32.251;
   1:L PR[91] R[100]mm/sec CNT100;
   1:  PR[GP1:91,1] = PR[GP1:90,1] + 3.141;
   1:  PR[GP1:91,2] = PR[GP1:90,2] + 32.133;
   1:L PR[91] R[100]mm/sec CNT100;
   1:  PR[GP1:91,1] = PR[GP1:90,1] + 1.940;
   1:  PR[GP1:91,2] = PR[GP1:90,2] + 31.464;
   1:L PR[91] R[100]mm/sec CNT100;
   1:  ! -- Layer/Ebene 109 -- !;
   1:  PR[91] = PR[90];
   1:  PR[GP1:91,1] = PR[GP1:90,1] + -1.658;
   1:  PR[GP1:91,2] = PR[GP1:90,2] + 32.005;
   1:  PR[GP1:91,3] = PR[GP1:90,3] + 66.795;
   1:L PR[91] R[100]mm/sec CNT100;
   1:  PR[GP1:91,1] = PR[GP1:90,1] + -2.535;
   1:  PR[GP1:91,2] = PR[GP1:90,2] + 32.209;
   1:L PR[91] R[100]mm/sec CNT100;
   1:  PR[GP1:91,1] = PR[GP1:90,1] + -3.334;
   1:  PR[GP1:91,2] = PR[GP1:90,2] + 32.774;
   1:L PR[91] R[100]mm/sec CNT100;
   1:  PR[GP1:91,1] = PR[GP1:90,1] + -3.781;
   1:  PR[GP1:91,2] = PR[GP1:90,2] + 33.008;
   1:L PR[91] R[100]mm/sec CNT100;
   1:  PR[GP1:91,1] = PR[GP1:90,1] + -4.378;
   1:  PR[GP1:91,2] = PR[GP1:90,2] + 33.200;
   1:L PR[91] R[100]mm/sec CNT100;
   1:  PR[GP1:91,1] = PR[GP1:90,1] + -16.259;
   1:  PR[GP1:91,2] = PR[GP1:90,2] + 37.307;
   1:L PR[91] R[100]mm/sec CNT100;
   1:  PR[GP1:91,1] = PR[GP1:90,1] + -17.365;
   1:  PR[GP1:91,2] = PR[GP1:90,2] + 37.452;
   1:L PR[91] R[100]mm/sec CNT100;
   1:  PR[GP1:91,1] = PR[GP1:90,1] + -18.725;
   1:  PR[GP1:91,2] = PR[GP1:90,2] + 37.405;
   1:L PR[91] R[100]mm/sec CNT100;
   1:  PR[GP1:91,1] = PR[GP1:90,1] + -30.177;
   1:  PR[GP1:91,2] = PR[GP1:90,2] + 37.347;
   1:L PR[91] R[100]mm/sec CNT100;
   1:  PR[GP1:91,1] = PR[GP1:90,1] + -31.935;
   1:  PR[GP1:91,2] = PR[GP1:90,2] + 36.968;
   1:L PR[91] R[100]mm/sec CNT100;
   1:  PR[GP1:91,1] = PR[GP1:90,1] + -33.913;
   1:  PR[GP1:91,2] = PR[GP1:90,2] + 36.185;
   1:L PR[91] R[100]mm/sec CNT100;
   1:  PR[GP1:91,1] = PR[GP1:90,1] + -43.290;
   1:  PR[GP1:91,2] = PR[GP1:90,2] + 32.855;
   1:L PR[91] R[100]mm/sec CNT100;
   1:  PR[GP1:91,1] = PR[GP1:90,1] + -45.385;
   1:  PR[GP1:91,2] = PR[GP1:90,2] + 31.550;
   1:L PR[91] R[100]mm/sec CNT100;
   1:  PR[GP1:91,1] = PR[GP1:90,1] + -47.457;
   1:  PR[GP1:91,2] = PR[GP1:90,2] + 29.711;
   1:L PR[91] R[100]mm/sec CNT100;
   1:  PR[GP1:91,1] = PR[GP1:90,1] + -54.021;
   1:  PR[GP1:91,2] = PR[GP1:90,2] + 24.398;
   1:L PR[91] R[100]mm/sec CNT100;
   1:  PR[GP1:91,1] = PR[GP1:90,1] + -55.816;
   1:  PR[GP1:91,2] = PR[GP1:90,2] + 22.063;
   1:L PR[91] R[100]mm/sec CNT100;
   1:  PR[GP1:91,1] = PR[GP1:90,1] + -57.345;
   1:  PR[GP1:91,2] = PR[GP1:90,2] + 19.096;
   1:L PR[91] R[100]mm/sec CNT100;
   1:  PR[GP1:91,1] = PR[GP1:90,1] + -61.093;
   1:  PR[GP1:91,2] = PR[GP1:90,2] + 12.835;
   1:L PR[91] R[100]mm/sec CNT100;
   1:  PR[GP1:91,1] = PR[GP1:90,1] + -61.994;
   1:  PR[GP1:91,2] = PR[GP1:90,2] + 9.777;
   1:L PR[91] R[100]mm/sec CNT100;
   1:  PR[GP1:91,1] = PR[GP1:90,1] + -62.296;
   1:  PR[GP1:91,2] = PR[GP1:90,2] + 6.483;
   1:L PR[91] R[100]mm/sec CNT100;
   1:  PR[GP1:91,1] = PR[GP1:90,1] + -63.509;
   1:  PR[GP1:91,2] = PR[GP1:90,2] + -0.100;
   1:L PR[91] R[100]mm/sec CNT100;
   1:  PR[GP1:91,1] = PR[GP1:90,1] + -63.214;
   1:  PR[GP1:91,2] = PR[GP1:90,2] + -3.362;
   1:L PR[91] R[100]mm/sec CNT100;
   1:  PR[GP1:91,1] = PR[GP1:90,1] + -62.001;
   1:  PR[GP1:91,2] = PR[GP1:90,2] + -9.896;
   1:L PR[91] R[100]mm/sec CNT100;
   1:  PR[GP1:91,1] = PR[GP1:90,1] + -61.086;
   1:  PR[GP1:91,2] = PR[GP1:90,2] + -13.000;
   1:L PR[91] R[100]mm/sec CNT100;
   1:  PR[GP1:91,1] = PR[GP1:90,1] + -59.604;
   1:  PR[GP1:91,2] = PR[GP1:90,2] + -15.906;
   1:L PR[91] R[100]mm/sec CNT100;
   1:  PR[GP1:91,1] = PR[GP1:90,1] + -55.824;
   1:  PR[GP1:91,2] = PR[GP1:90,2] + -22.195;
   1:L PR[91] R[100]mm/sec CNT100;
   1:  PR[GP1:91,1] = PR[GP1:90,1] + -54.009;
   1:  PR[GP1:91,2] = PR[GP1:90,2] + -24.558;
   1:L PR[91] R[100]mm/sec CNT100;
   1:  PR[GP1:91,1] = PR[GP1:90,1] + -51.966;
   1:  PR[GP1:91,2] = PR[GP1:90,2] + -26.391;
   1:L PR[91] R[100]mm/sec CNT100;
   1:  PR[GP1:91,1] = PR[GP1:90,1] + -45.390;
   1:  PR[GP1:91,2] = PR[GP1:90,2] + -31.691;
   1:L PR[91] R[100]mm/sec CNT100;
   1:  PR[GP1:91,1] = PR[GP1:90,1] + -43.272;
   1:  PR[GP1:91,2] = PR[GP1:90,2] + -33.010;
   1:L PR[91] R[100]mm/sec CNT100;
   1:  PR[GP1:91,1] = PR[GP1:90,1] + -41.196;
   1:  PR[GP1:91,2] = PR[GP1:90,2] + -33.844;
   1:L PR[91] R[100]mm/sec CNT100;
   1:  PR[GP1:91,1] = PR[GP1:90,1] + -31.933;
   1:  PR[GP1:91,2] = PR[GP1:90,2] + -37.112;
   1:L PR[91] R[100]mm/sec CNT100;
   1:  PR[GP1:91,1] = PR[GP1:90,1] + -30.154;
   1:  PR[GP1:91,2] = PR[GP1:90,2] + -37.496;
   1:L PR[91] R[100]mm/sec CNT100;
   1:  PR[GP1:91,1] = PR[GP1:90,1] + -28.532;
   1:  PR[GP1:91,2] = PR[GP1:90,2] + -37.558;
   1:L PR[91] R[100]mm/sec CNT100;
   1:  PR[GP1:91,1] = PR[GP1:90,1] + -17.355;
   1:  PR[GP1:91,2] = PR[GP1:90,2] + -37.594;
   1:L PR[91] R[100]mm/sec CNT100;
   1:  PR[GP1:91,1] = PR[GP1:90,1] + -16.233;
   1:  PR[GP1:91,2] = PR[GP1:90,2] + -37.447;
   1:L PR[91] R[100]mm/sec CNT100;
   1:  PR[GP1:91,1] = PR[GP1:90,1] + -15.257;
   1:  PR[GP1:91,2] = PR[GP1:90,2] + -37.137;
   1:L PR[91] R[100]mm/sec CNT100;
   1:  PR[GP1:91,1] = PR[GP1:90,1] + -3.768;
   1:  PR[GP1:91,2] = PR[GP1:90,2] + -33.144;
   1:L PR[91] R[100]mm/sec CNT100;
   1:  PR[GP1:91,1] = PR[GP1:90,1] + -3.326;
   1:  PR[GP1:91,2] = PR[GP1:90,2] + -32.913;
   1:L PR[91] R[100]mm/sec CNT100;
   1:  PR[GP1:91,1] = PR[GP1:90,1] + -2.491;
   1:  PR[GP1:91,2] = PR[GP1:90,2] + -32.306;
   1:L PR[91] R[100]mm/sec CNT100;
   1:  PR[GP1:91,1] = PR[GP1:90,1] + 0.251;
   1:  PR[GP1:91,2] = PR[GP1:90,2] + -32.196;
   1:L PR[91] R[100]mm/sec CNT100;
   1:  PR[GP1:91,1] = PR[GP1:90,1] + 1.998;
   1:  PR[GP1:91,2] = PR[GP1:90,2] + -31.824;
   1:L PR[91] R[100]mm/sec CNT100;
   1:  PR[GP1:91,1] = PR[GP1:90,1] + 2.513;
   1:  PR[GP1:91,2] = PR[GP1:90,2] + -32.238;
   1:L PR[91] R[100]mm/sec CNT100;
   1:  PR[GP1:91,1] = PR[GP1:90,1] + 2.803;
   1:  PR[GP1:91,2] = PR[GP1:90,2] + -32.383;
   1:L PR[91] R[100]mm/sec CNT100;
   1:  PR[GP1:91,1] = PR[GP1:90,1] + 3.534;
   1:  PR[GP1:91,2] = PR[GP1:90,2] + -32.913;
   1:L PR[91] R[100]mm/sec CNT100;
   1:  PR[GP1:91,1] = PR[GP1:90,1] + 3.965;
   1:  PR[GP1:91,2] = PR[GP1:90,2] + -33.139;
   1:L PR[91] R[100]mm/sec CNT100;
   1:  PR[GP1:91,1] = PR[GP1:90,1] + 4.554;
   1:  PR[GP1:91,2] = PR[GP1:90,2] + -33.328;
   1:L PR[91] R[100]mm/sec CNT100;
   1:  PR[GP1:91,1] = PR[GP1:90,1] + 16.450;
   1:  PR[GP1:91,2] = PR[GP1:90,2] + -37.447;
   1:L PR[91] R[100]mm/sec CNT100;
   1:  PR[GP1:91,1] = PR[GP1:90,1] + 17.554;
   1:  PR[GP1:91,2] = PR[GP1:90,2] + -37.592;
   1:L PR[91] R[100]mm/sec CNT100;
   1:  PR[GP1:91,1] = PR[GP1:90,1] + 18.906;
   1:  PR[GP1:91,2] = PR[GP1:90,2] + -37.546;
   1:L PR[91] R[100]mm/sec CNT100;
   1:  PR[GP1:91,1] = PR[GP1:90,1] + 30.364;
   1:  PR[GP1:91,2] = PR[GP1:90,2] + -37.496;
   1:L PR[91] R[100]mm/sec CNT100;
   1:  PR[GP1:91,1] = PR[GP1:90,1] + 32.119;
   1:  PR[GP1:91,2] = PR[GP1:90,2] + -37.118;
   1:L PR[91] R[100]mm/sec CNT100;
   1:  PR[GP1:91,1] = PR[GP1:90,1] + 34.100;
   1:  PR[GP1:91,2] = PR[GP1:90,2] + -36.338;
   1:L PR[91] R[100]mm/sec CNT100;
   1:  PR[GP1:91,1] = PR[GP1:90,1] + 43.483;
   1:  PR[GP1:91,2] = PR[GP1:90,2] + -33.012;
   1:L PR[91] R[100]mm/sec CNT100;
   1:  PR[GP1:91,1] = PR[GP1:90,1] + 45.564;
   1:  PR[GP1:91,2] = PR[GP1:90,2] + -31.722;
   1:L PR[91] R[100]mm/sec CNT100;
   1:  PR[GP1:91,1] = PR[GP1:90,1] + 47.624;
   1:  PR[GP1:91,2] = PR[GP1:90,2] + -29.898;
   1:L PR[91] R[100]mm/sec CNT100;
   1:  PR[GP1:91,1] = PR[GP1:90,1] + 54.194;
   1:  PR[GP1:91,2] = PR[GP1:90,2] + -24.580;
   1:L PR[91] R[100]mm/sec CNT100;
   1:  PR[GP1:91,1] = PR[GP1:90,1] + 56.007;
   1:  PR[GP1:91,2] = PR[GP1:90,2] + -22.226;
   1:L PR[91] R[100]mm/sec CNT100;
   1:  PR[GP1:91,1] = PR[GP1:90,1] + 57.541;
   1:  PR[GP1:91,2] = PR[GP1:90,2] + -19.283;
   1:L PR[91] R[100]mm/sec CNT100;
   1:  PR[GP1:91,1] = PR[GP1:90,1] + 61.292;
   1:  PR[GP1:91,2] = PR[GP1:90,2] + -13.034;
   1:L PR[91] R[100]mm/sec CNT100;
   1:  PR[GP1:91,1] = PR[GP1:90,1] + 62.192;
   1:  PR[GP1:91,2] = PR[GP1:90,2] + -10.022;
   1:L PR[91] R[100]mm/sec CNT100;
   1:  PR[GP1:91,1] = PR[GP1:90,1] + 62.508;
   1:  PR[GP1:91,2] = PR[GP1:90,2] + -6.637;
   1:L PR[91] R[100]mm/sec CNT100;
   1:  PR[GP1:91,1] = PR[GP1:90,1] + 63.722;
   1:  PR[GP1:91,2] = PR[GP1:90,2] + -0.045;
   1:L PR[91] R[100]mm/sec CNT100;
   1:  PR[GP1:91,1] = PR[GP1:90,1] + 63.412;
   1:  PR[GP1:91,2] = PR[GP1:90,2] + 3.309;
   1:L PR[91] R[100]mm/sec CNT100;
   1:  PR[GP1:91,1] = PR[GP1:90,1] + 62.200;
   1:  PR[GP1:91,2] = PR[GP1:90,2] + 9.850;
   1:L PR[91] R[100]mm/sec CNT100;
   1:  PR[GP1:91,1] = PR[GP1:90,1] + 61.287;
   1:  PR[GP1:91,2] = PR[GP1:90,2] + 12.906;
   1:L PR[91] R[100]mm/sec CNT100;
   1:  PR[GP1:91,1] = PR[GP1:90,1] + 59.801;
   1:  PR[GP1:91,2] = PR[GP1:90,2] + 15.787;
   1:L PR[91] R[100]mm/sec CNT100;
   1:  PR[GP1:91,1] = PR[GP1:90,1] + 56.022;
   1:  PR[GP1:91,2] = PR[GP1:90,2] + 22.064;
   1:L PR[91] R[100]mm/sec CNT100;
   1:  PR[GP1:91,1] = PR[GP1:90,1] + 54.188;
   1:  PR[GP1:91,2] = PR[GP1:90,2] + 24.444;
   1:L PR[91] R[100]mm/sec CNT100;
   1:  PR[GP1:91,1] = PR[GP1:90,1] + 52.156;
   1:  PR[GP1:91,2] = PR[GP1:90,2] + 26.261;
   1:L PR[91] R[100]mm/sec CNT100;
   1:  PR[GP1:91,1] = PR[GP1:90,1] + 45.583;
   1:  PR[GP1:91,2] = PR[GP1:90,2] + 31.567;
   1:L PR[91] R[100]mm/sec CNT100;
   1:  PR[GP1:91,1] = PR[GP1:90,1] + 43.480;
   1:  PR[GP1:91,2] = PR[GP1:90,2] + 32.870;
   1:L PR[91] R[100]mm/sec CNT100;
   1:  PR[GP1:91,1] = PR[GP1:90,1] + 41.401;
   1:  PR[GP1:91,2] = PR[GP1:90,2] + 33.701;
   1:L PR[91] R[100]mm/sec CNT100;
   1:  PR[GP1:91,1] = PR[GP1:90,1] + 32.143;
   1:  PR[GP1:91,2] = PR[GP1:90,2] + 36.970;
   1:L PR[91] R[100]mm/sec CNT100;
   1:  PR[GP1:91,1] = PR[GP1:90,1] + 30.367;
   1:  PR[GP1:91,2] = PR[GP1:90,2] + 37.352;
   1:L PR[91] R[100]mm/sec CNT100;
   1:  PR[GP1:91,1] = PR[GP1:90,1] + 28.753;
   1:  PR[GP1:91,2] = PR[GP1:90,2] + 37.413;
   1:L PR[91] R[100]mm/sec CNT100;
   1:  PR[GP1:91,1] = PR[GP1:90,1] + 17.581;
   1:  PR[GP1:91,2] = PR[GP1:90,2] + 37.452;
   1:L PR[91] R[100]mm/sec CNT100;
   1:  PR[GP1:91,1] = PR[GP1:90,1] + 16.461;
   1:  PR[GP1:91,2] = PR[GP1:90,2] + 37.305;
   1:L PR[91] R[100]mm/sec CNT100;
   1:  PR[GP1:91,1] = PR[GP1:90,1] + 15.483;
   1:  PR[GP1:91,2] = PR[GP1:90,2] + 36.994;
   1:L PR[91] R[100]mm/sec CNT100;
   1:  PR[GP1:91,1] = PR[GP1:90,1] + 3.990;
   1:  PR[GP1:91,2] = PR[GP1:90,2] + 33.009;
   1:L PR[91] R[100]mm/sec CNT100;
   1:  PR[GP1:91,1] = PR[GP1:90,1] + 3.541;
   1:  PR[GP1:91,2] = PR[GP1:90,2] + 32.775;
   1:L PR[91] R[100]mm/sec CNT100;
   1:  PR[GP1:91,1] = PR[GP1:90,1] + 3.107;
   1:  PR[GP1:91,2] = PR[GP1:90,2] + 32.468;
   1:L PR[91] R[100]mm/sec CNT100;
   1:  PR[GP1:91,1] = PR[GP1:90,1] + 3.113;
   1:  PR[GP1:91,2] = PR[GP1:90,2] + 32.344;
   1:L PR[91] R[100]mm/sec CNT100;
   1:  PR[GP1:91,1] = PR[GP1:90,1] + 1.970;
   1:  PR[GP1:91,2] = PR[GP1:90,2] + 31.707;
   1:L PR[91] R[100]mm/sec CNT100;
   1:  ! -- Layer/Ebene 110 -- !;
   1:  PR[91] = PR[90];
   1:  PR[GP1:91,1] = PR[GP1:90,1] + -1.809;
   1:  PR[GP1:91,2] = PR[GP1:90,2] + 32.264;
   1:  PR[GP1:91,3] = PR[GP1:90,3] + 67.405;
   1:L PR[91] R[100]mm/sec CNT100;
   1:  PR[GP1:91,1] = PR[GP1:90,1] + -2.507;
   1:  PR[GP1:91,2] = PR[GP1:90,2] + 32.426;
   1:L PR[91] R[100]mm/sec CNT100;
   1:  PR[GP1:91,1] = PR[GP1:90,1] + -3.123;
   1:  PR[GP1:91,2] = PR[GP1:90,2] + 32.861;
   1:L PR[91] R[100]mm/sec CNT100;
   1:  PR[GP1:91,1] = PR[GP1:90,1] + -3.439;
   1:  PR[GP1:91,2] = PR[GP1:90,2] + 33.026;
   1:L PR[91] R[100]mm/sec CNT100;
   1:  PR[GP1:91,1] = PR[GP1:90,1] + -3.877;
   1:  PR[GP1:91,2] = PR[GP1:90,2] + 33.167;
   1:L PR[91] R[100]mm/sec CNT100;
   1:  PR[GP1:91,1] = PR[GP1:90,1] + -16.061;
   1:  PR[GP1:91,2] = PR[GP1:90,2] + 37.379;
   1:L PR[91] R[100]mm/sec CNT100;
   1:  PR[GP1:91,1] = PR[GP1:90,1] + -17.013;
   1:  PR[GP1:91,2] = PR[GP1:90,2] + 37.504;
   1:L PR[91] R[100]mm/sec CNT100;
   1:  PR[GP1:91,1] = PR[GP1:90,1] + -18.197;
   1:  PR[GP1:91,2] = PR[GP1:90,2] + 37.463;
   1:L PR[91] R[100]mm/sec CNT100;
   1:  PR[GP1:91,1] = PR[GP1:90,1] + -29.989;
   1:  PR[GP1:91,2] = PR[GP1:90,2] + 37.404;
   1:L PR[91] R[100]mm/sec CNT100;
   1:  PR[GP1:91,1] = PR[GP1:90,1] + -31.589;
   1:  PR[GP1:91,2] = PR[GP1:90,2] + 37.059;
   1:L PR[91] R[100]mm/sec CNT100;
   1:  PR[GP1:91,1] = PR[GP1:90,1] + -33.398;
   1:  PR[GP1:91,2] = PR[GP1:90,2] + 36.343;
   1:L PR[91] R[100]mm/sec CNT100;
   1:  PR[GP1:91,1] = PR[GP1:90,1] + -43.107;
   1:  PR[GP1:91,2] = PR[GP1:90,2] + 32.895;
   1:L PR[91] R[100]mm/sec CNT100;
   1:  PR[GP1:91,1] = PR[GP1:90,1] + -45.060;
   1:  PR[GP1:91,2] = PR[GP1:90,2] + 31.678;
   1:L PR[91] R[100]mm/sec CNT100;
   1:  PR[GP1:91,1] = PR[GP1:90,1] + -46.996;
   1:  PR[GP1:91,2] = PR[GP1:90,2] + 29.959;
   1:L PR[91] R[100]mm/sec CNT100;
   1:  PR[GP1:91,1] = PR[GP1:90,1] + -53.838;
   1:  PR[GP1:91,2] = PR[GP1:90,2] + 24.423;
   1:L PR[91] R[100]mm/sec CNT100;
   1:  PR[GP1:91,1] = PR[GP1:90,1] + -55.531;
   1:  PR[GP1:91,2] = PR[GP1:90,2] + 22.219;
   1:L PR[91] R[100]mm/sec CNT100;
   1:  PR[GP1:91,1] = PR[GP1:90,1] + -56.977;
   1:  PR[GP1:91,2] = PR[GP1:90,2] + 19.414;
   1:L PR[91] R[100]mm/sec CNT100;
   1:  PR[GP1:91,1] = PR[GP1:90,1] + -60.906;
   1:  PR[GP1:91,2] = PR[GP1:90,2] + 12.850;
   1:L PR[91] R[100]mm/sec CNT100;
   1:  PR[GP1:91,1] = PR[GP1:90,1] + -61.761;
   1:  PR[GP1:91,2] = PR[GP1:90,2] + 9.949;
   1:L PR[91] R[100]mm/sec CNT100;
   1:  PR[GP1:91,1] = PR[GP1:90,1] + -62.048;
   1:  PR[GP1:91,2] = PR[GP1:90,2] + 6.817;
   1:L PR[91] R[100]mm/sec CNT100;
   1:  PR[GP1:91,1] = PR[GP1:90,1] + -63.323;
   1:  PR[GP1:91,2] = PR[GP1:90,2] + -0.100;
   1:L PR[91] R[100]mm/sec CNT100;
   1:  PR[GP1:91,1] = PR[GP1:90,1] + -63.042;
   1:  PR[GP1:91,2] = PR[GP1:90,2] + -3.206;
   1:L PR[91] R[100]mm/sec CNT100;
   1:  PR[GP1:91,1] = PR[GP1:90,1] + -61.768;
   1:  PR[GP1:91,2] = PR[GP1:90,2] + -10.068;
   1:L PR[91] R[100]mm/sec CNT100;
   1:  PR[GP1:91,1] = PR[GP1:90,1] + -60.899;
   1:  PR[GP1:91,2] = PR[GP1:90,2] + -13.016;
   1:L PR[91] R[100]mm/sec CNT100;
   1:  PR[GP1:91,1] = PR[GP1:90,1] + -59.492;
   1:  PR[GP1:91,2] = PR[GP1:90,2] + -15.776;
   1:L PR[91] R[100]mm/sec CNT100;
   1:  PR[GP1:91,1] = PR[GP1:90,1] + -55.539;
   1:  PR[GP1:91,2] = PR[GP1:90,2] + -22.351;
   1:L PR[91] R[100]mm/sec CNT100;
   1:  PR[GP1:91,1] = PR[GP1:90,1] + -53.825;
   1:  PR[GP1:91,2] = PR[GP1:90,2] + -24.583;
   1:L PR[91] R[100]mm/sec CNT100;
   1:  PR[GP1:91,1] = PR[GP1:90,1] + -51.896;
   1:  PR[GP1:91,2] = PR[GP1:90,2] + -26.313;
   1:L PR[91] R[100]mm/sec CNT100;
   1:  PR[GP1:91,1] = PR[GP1:90,1] + -45.064;
   1:  PR[GP1:91,2] = PR[GP1:90,2] + -31.819;
   1:L PR[91] R[100]mm/sec CNT100;
   1:  PR[GP1:91,1] = PR[GP1:90,1] + -43.088;
   1:  PR[GP1:91,2] = PR[GP1:90,2] + -33.050;
   1:L PR[91] R[100]mm/sec CNT100;
   1:  PR[GP1:91,1] = PR[GP1:90,1] + -41.150;
   1:  PR[GP1:91,2] = PR[GP1:90,2] + -33.829;
   1:L PR[91] R[100]mm/sec CNT100;
   1:  PR[GP1:91,1] = PR[GP1:90,1] + -31.587;
   1:  PR[GP1:91,2] = PR[GP1:90,2] + -37.203;
   1:L PR[91] R[100]mm/sec CNT100;
   1:  PR[GP1:91,1] = PR[GP1:90,1] + -29.965;
   1:  PR[GP1:91,2] = PR[GP1:90,2] + -37.553;
   1:L PR[91] R[100]mm/sec CNT100;
   1:  PR[GP1:91,1] = PR[GP1:90,1] + -28.486;
   1:  PR[GP1:91,2] = PR[GP1:90,2] + -37.609;
   1:L PR[91] R[100]mm/sec CNT100;
   1:  PR[GP1:91,1] = PR[GP1:90,1] + -17.003;
   1:  PR[GP1:91,2] = PR[GP1:90,2] + -37.646;
   1:L PR[91] R[100]mm/sec CNT100;
   1:  PR[GP1:91,1] = PR[GP1:90,1] + -16.034;
   1:  PR[GP1:91,2] = PR[GP1:90,2] + -37.519;
   1:L PR[91] R[100]mm/sec CNT100;
   1:  PR[GP1:91,1] = PR[GP1:90,1] + -15.189;
   1:  PR[GP1:91,2] = PR[GP1:90,2] + -37.250;
   1:L PR[91] R[100]mm/sec CNT100;
   1:  PR[GP1:91,1] = PR[GP1:90,1] + -3.425;
   1:  PR[GP1:91,2] = PR[GP1:90,2] + -33.162;
   1:L PR[91] R[100]mm/sec CNT100;
   1:  PR[GP1:91,1] = PR[GP1:90,1] + -3.116;
   1:  PR[GP1:91,2] = PR[GP1:90,2] + -33.000;
   1:L PR[91] R[100]mm/sec CNT100;
   1:  PR[GP1:91,1] = PR[GP1:90,1] + -2.463;
   1:  PR[GP1:91,2] = PR[GP1:90,2] + -32.526;
   1:L PR[91] R[100]mm/sec CNT100;
   1:  PR[GP1:91,1] = PR[GP1:90,1] + 0.417;
   1:  PR[GP1:91,2] = PR[GP1:90,2] + -32.411;
   1:L PR[91] R[100]mm/sec CNT100;
   1:  PR[GP1:91,1] = PR[GP1:90,1] + 2.028;
   1:  PR[GP1:91,2] = PR[GP1:90,2] + -32.067;
   1:L PR[91] R[100]mm/sec CNT100;
   1:  PR[GP1:91,1] = PR[GP1:90,1] + 2.562;
   1:  PR[GP1:91,2] = PR[GP1:90,2] + -32.497;
   1:L PR[91] R[100]mm/sec CNT100;
   1:  PR[GP1:91,1] = PR[GP1:90,1] + 2.775;
   1:  PR[GP1:91,2] = PR[GP1:90,2] + -32.603;
   1:L PR[91] R[100]mm/sec CNT100;
   1:  PR[GP1:91,1] = PR[GP1:90,1] + 3.322;
   1:  PR[GP1:91,2] = PR[GP1:90,2] + -33.000;
   1:L PR[91] R[100]mm/sec CNT100;
   1:  PR[GP1:91,1] = PR[GP1:90,1] + 3.623;
   1:  PR[GP1:91,2] = PR[GP1:90,2] + -33.157;
   1:L PR[91] R[100]mm/sec CNT100;
   1:  PR[GP1:91,1] = PR[GP1:90,1] + 4.052;
   1:  PR[GP1:91,2] = PR[GP1:90,2] + -33.295;
   1:L PR[91] R[100]mm/sec CNT100;
   1:  PR[GP1:91,1] = PR[GP1:90,1] + 16.251;
   1:  PR[GP1:91,2] = PR[GP1:90,2] + -37.519;
   1:L PR[91] R[100]mm/sec CNT100;
   1:  PR[GP1:91,1] = PR[GP1:90,1] + 17.202;
   1:  PR[GP1:91,2] = PR[GP1:90,2] + -37.644;
   1:L PR[91] R[100]mm/sec CNT100;
   1:  PR[GP1:91,1] = PR[GP1:90,1] + 18.379;
   1:  PR[GP1:91,2] = PR[GP1:90,2] + -37.604;
   1:L PR[91] R[100]mm/sec CNT100;
   1:  PR[GP1:91,1] = PR[GP1:90,1] + 30.176;
   1:  PR[GP1:91,2] = PR[GP1:90,2] + -37.552;
   1:L PR[91] R[100]mm/sec CNT100;
   1:  PR[GP1:91,1] = PR[GP1:90,1] + 31.774;
   1:  PR[GP1:91,2] = PR[GP1:90,2] + -37.209;
   1:L PR[91] R[100]mm/sec CNT100;
   1:  PR[GP1:91,1] = PR[GP1:90,1] + 33.584;
   1:  PR[GP1:91,2] = PR[GP1:90,2] + -36.495;
   1:L PR[91] R[100]mm/sec CNT100;
   1:  PR[GP1:91,1] = PR[GP1:90,1] + 43.300;
   1:  PR[GP1:91,2] = PR[GP1:90,2] + -33.052;
   1:L PR[91] R[100]mm/sec CNT100;
   1:  PR[GP1:91,1] = PR[GP1:90,1] + 45.241;
   1:  PR[GP1:91,2] = PR[GP1:90,2] + -31.849;
   1:L PR[91] R[100]mm/sec CNT100;
   1:  PR[GP1:91,1] = PR[GP1:90,1] + 47.166;
   1:  PR[GP1:91,2] = PR[GP1:90,2] + -30.145;
   1:L PR[91] R[100]mm/sec CNT100;
   1:  PR[GP1:91,1] = PR[GP1:90,1] + 54.012;
   1:  PR[GP1:91,2] = PR[GP1:90,2] + -24.602;
   1:L PR[91] R[100]mm/sec CNT100;
   1:  PR[GP1:91,1] = PR[GP1:90,1] + 55.724;
   1:  PR[GP1:91,2] = PR[GP1:90,2] + -22.381;
   1:L PR[91] R[100]mm/sec CNT100;
   1:  PR[GP1:91,1] = PR[GP1:90,1] + 57.173;
   1:  PR[GP1:91,2] = PR[GP1:90,2] + -19.599;
   1:L PR[91] R[100]mm/sec CNT100;
   1:  PR[GP1:91,1] = PR[GP1:90,1] + 61.105;
   1:  PR[GP1:91,2] = PR[GP1:90,2] + -13.048;
   1:L PR[91] R[100]mm/sec CNT100;
   1:  PR[GP1:91,1] = PR[GP1:90,1] + 61.959;
   1:  PR[GP1:91,2] = PR[GP1:90,2] + -10.190;
   1:L PR[91] R[100]mm/sec CNT100;
   1:  PR[GP1:91,1] = PR[GP1:90,1] + 62.260;
   1:  PR[GP1:91,2] = PR[GP1:90,2] + -6.972;
   1:L PR[91] R[100]mm/sec CNT100;
   1:  PR[GP1:91,1] = PR[GP1:90,1] + 63.536;
   1:  PR[GP1:91,2] = PR[GP1:90,2] + -0.045;
   1:L PR[91] R[100]mm/sec CNT100;
   1:  PR[GP1:91,1] = PR[GP1:90,1] + 63.241;
   1:  PR[GP1:91,2] = PR[GP1:90,2] + 3.149;
   1:L PR[91] R[100]mm/sec CNT100;
   1:  PR[GP1:91,1] = PR[GP1:90,1] + 61.968;
   1:  PR[GP1:91,2] = PR[GP1:90,2] + 10.017;
   1:L PR[91] R[100]mm/sec CNT100;
   1:  PR[GP1:91,1] = PR[GP1:90,1] + 61.101;
   1:  PR[GP1:91,2] = PR[GP1:90,2] + 12.920;
   1:L PR[91] R[100]mm/sec CNT100;
   1:  PR[GP1:91,1] = PR[GP1:90,1] + 59.689;
   1:  PR[GP1:91,2] = PR[GP1:90,2] + 15.656;
   1:L PR[91] R[100]mm/sec CNT100;
   1:  PR[GP1:91,1] = PR[GP1:90,1] + 55.738;
   1:  PR[GP1:91,2] = PR[GP1:90,2] + 22.218;
   1:L PR[91] R[100]mm/sec CNT100;
   1:  PR[GP1:91,1] = PR[GP1:90,1] + 54.006;
   1:  PR[GP1:91,2] = PR[GP1:90,2] + 24.466;
   1:L PR[91] R[100]mm/sec CNT100;
   1:  PR[GP1:91,1] = PR[GP1:90,1] + 52.087;
   1:  PR[GP1:91,2] = PR[GP1:90,2] + 26.182;
   1:L PR[91] R[100]mm/sec CNT100;
   1:  PR[GP1:91,1] = PR[GP1:90,1] + 45.260;
   1:  PR[GP1:91,2] = PR[GP1:90,2] + 31.694;
   1:L PR[91] R[100]mm/sec CNT100;
   1:  PR[GP1:91,1] = PR[GP1:90,1] + 43.297;
   1:  PR[GP1:91,2] = PR[GP1:90,2] + 32.910;
   1:L PR[91] R[100]mm/sec CNT100;
   1:  PR[GP1:91,1] = PR[GP1:90,1] + 41.356;
   1:  PR[GP1:91,2] = PR[GP1:90,2] + 33.685;
   1:L PR[91] R[100]mm/sec CNT100;
   1:  PR[GP1:91,1] = PR[GP1:90,1] + 31.798;
   1:  PR[GP1:91,2] = PR[GP1:90,2] + 37.060;
   1:L PR[91] R[100]mm/sec CNT100;
   1:  PR[GP1:91,1] = PR[GP1:90,1] + 30.180;
   1:  PR[GP1:91,2] = PR[GP1:90,2] + 37.408;
   1:L PR[91] R[100]mm/sec CNT100;
   1:  PR[GP1:91,1] = PR[GP1:90,1] + 28.707;
   1:  PR[GP1:91,2] = PR[GP1:90,2] + 37.464;
   1:L PR[91] R[100]mm/sec CNT100;
   1:  PR[GP1:91,1] = PR[GP1:90,1] + 17.230;
   1:  PR[GP1:91,2] = PR[GP1:90,2] + 37.504;
   1:L PR[91] R[100]mm/sec CNT100;
   1:  PR[GP1:91,1] = PR[GP1:90,1] + 16.262;
   1:  PR[GP1:91,2] = PR[GP1:90,2] + 37.377;
   1:L PR[91] R[100]mm/sec CNT100;
   1:  PR[GP1:91,1] = PR[GP1:90,1] + 15.416;
   1:  PR[GP1:91,2] = PR[GP1:90,2] + 37.107;
   1:L PR[91] R[100]mm/sec CNT100;
   1:  PR[GP1:91,1] = PR[GP1:90,1] + 3.649;
   1:  PR[GP1:91,2] = PR[GP1:90,2] + 33.028;
   1:L PR[91] R[100]mm/sec CNT100;
   1:  PR[GP1:91,1] = PR[GP1:90,1] + 3.330;
   1:  PR[GP1:91,2] = PR[GP1:90,2] + 32.861;
   1:L PR[91] R[100]mm/sec CNT100;
   1:  PR[GP1:91,1] = PR[GP1:90,1] + 3.079;
   1:  PR[GP1:91,2] = PR[GP1:90,2] + 32.684;
   1:L PR[91] R[100]mm/sec CNT100;
   1:  PR[GP1:91,1] = PR[GP1:90,1] + 3.085;
   1:  PR[GP1:91,2] = PR[GP1:90,2] + 32.555;
   1:L PR[91] R[100]mm/sec CNT100;
   1:  PR[GP1:91,1] = PR[GP1:90,1] + 2.000;
   1:  PR[GP1:91,2] = PR[GP1:90,2] + 31.951;
   1:L PR[91] R[100]mm/sec CNT100;
   1:  ! -- Layer/Ebene 111 -- !;
   1:  PR[91] = PR[90];
   1:  PR[GP1:91,1] = PR[GP1:90,1] + -1.960;
   1:  PR[GP1:91,2] = PR[GP1:90,2] + 32.522;
   1:  PR[GP1:91,3] = PR[GP1:90,3] + 68.015;
   1:L PR[91] R[100]mm/sec CNT100;
   1:  PR[GP1:91,1] = PR[GP1:90,1] + -2.479;
   1:  PR[GP1:91,2] = PR[GP1:90,2] + 32.642;
   1:L PR[91] R[100]mm/sec CNT100;
   1:  PR[GP1:91,1] = PR[GP1:90,1] + -2.913;
   1:  PR[GP1:91,2] = PR[GP1:90,2] + 32.949;
   1:L PR[91] R[100]mm/sec CNT100;
   1:  PR[GP1:91,1] = PR[GP1:90,1] + -3.103;
   1:  PR[GP1:91,2] = PR[GP1:90,2] + 33.048;
   1:L PR[91] R[100]mm/sec CNT100;
   1:  PR[GP1:91,1] = PR[GP1:90,1] + -15.862;
   1:  PR[GP1:91,2] = PR[GP1:90,2] + 37.452;
   1:L PR[91] R[100]mm/sec CNT100;
   1:  PR[GP1:91,1] = PR[GP1:90,1] + -16.662;
   1:  PR[GP1:91,2] = PR[GP1:90,2] + 37.556;
   1:L PR[91] R[100]mm/sec CNT100;
   1:  PR[GP1:91,1] = PR[GP1:90,1] + -17.669;
   1:  PR[GP1:91,2] = PR[GP1:90,2] + 37.521;
   1:L PR[91] R[100]mm/sec CNT100;
   1:  PR[GP1:91,1] = PR[GP1:90,1] + -29.801;
   1:  PR[GP1:91,2] = PR[GP1:90,2] + 37.461;
   1:L PR[91] R[100]mm/sec CNT100;
   1:  PR[GP1:91,1] = PR[GP1:90,1] + -31.244;
   1:  PR[GP1:91,2] = PR[GP1:90,2] + 37.149;
   1:L PR[91] R[100]mm/sec CNT100;
   1:  PR[GP1:91,1] = PR[GP1:90,1] + -32.882;
   1:  PR[GP1:91,2] = PR[GP1:90,2] + 36.501;
   1:L PR[91] R[100]mm/sec CNT100;
   1:  PR[GP1:91,1] = PR[GP1:90,1] + -42.923;
   1:  PR[GP1:91,2] = PR[GP1:90,2] + 32.935;
   1:L PR[91] R[100]mm/sec CNT100;
   1:  PR[GP1:91,1] = PR[GP1:90,1] + -44.735;
   1:  PR[GP1:91,2] = PR[GP1:90,2] + 31.807;
   1:L PR[91] R[100]mm/sec CNT100;
   1:  PR[GP1:91,1] = PR[GP1:90,1] + -46.536;
   1:  PR[GP1:91,2] = PR[GP1:90,2] + 30.208;
   1:L PR[91] R[100]mm/sec CNT100;
   1:  PR[GP1:91,1] = PR[GP1:90,1] + -53.654;
   1:  PR[GP1:91,2] = PR[GP1:90,2] + 24.447;
   1:L PR[91] R[100]mm/sec CNT100;
   1:  PR[GP1:91,1] = PR[GP1:90,1] + -55.246;
   1:  PR[GP1:91,2] = PR[GP1:90,2] + 22.375;
   1:L PR[91] R[100]mm/sec CNT100;
   1:  PR[GP1:91,1] = PR[GP1:90,1] + -56.608;
   1:  PR[GP1:91,2] = PR[GP1:90,2] + 19.732;
   1:L PR[91] R[100]mm/sec CNT100;
   1:  PR[GP1:91,1] = PR[GP1:90,1] + -60.719;
   1:  PR[GP1:91,2] = PR[GP1:90,2] + 12.866;
   1:L PR[91] R[100]mm/sec CNT100;
   1:  PR[GP1:91,1] = PR[GP1:90,1] + -61.528;
   1:  PR[GP1:91,2] = PR[GP1:90,2] + 10.120;
   1:L PR[91] R[100]mm/sec CNT100;
   1:  PR[GP1:91,1] = PR[GP1:90,1] + -61.800;
   1:  PR[GP1:91,2] = PR[GP1:90,2] + 7.151;
   1:L PR[91] R[100]mm/sec CNT100;
   1:  PR[GP1:91,1] = PR[GP1:90,1] + -63.136;
   1:  PR[GP1:91,2] = PR[GP1:90,2] + -0.100;
   1:L PR[91] R[100]mm/sec CNT100;
   1:  PR[GP1:91,1] = PR[GP1:90,1] + -62.870;
   1:  PR[GP1:91,2] = PR[GP1:90,2] + -3.049;
   1:L PR[91] R[100]mm/sec CNT100;
   1:  PR[GP1:91,1] = PR[GP1:90,1] + -61.535;
   1:  PR[GP1:91,2] = PR[GP1:90,2] + -10.240;
   1:L PR[91] R[100]mm/sec CNT100;
   1:  PR[GP1:91,1] = PR[GP1:90,1] + -60.712;
   1:  PR[GP1:91,2] = PR[GP1:90,2] + -13.032;
   1:L PR[91] R[100]mm/sec CNT100;
   1:  PR[GP1:91,1] = PR[GP1:90,1] + -59.379;
   1:  PR[GP1:91,2] = PR[GP1:90,2] + -15.646;
   1:L PR[91] R[100]mm/sec CNT100;
   1:  PR[GP1:91,1] = PR[GP1:90,1] + -55.255;
   1:  PR[GP1:91,2] = PR[GP1:90,2] + -22.507;
   1:L PR[91] R[100]mm/sec CNT100;
   1:  PR[GP1:91,1] = PR[GP1:90,1] + -53.642;
   1:  PR[GP1:91,2] = PR[GP1:90,2] + -24.607;
   1:L PR[91] R[100]mm/sec CNT100;
   1:  PR[GP1:91,1] = PR[GP1:90,1] + -51.826;
   1:  PR[GP1:91,2] = PR[GP1:90,2] + -26.236;
   1:L PR[91] R[100]mm/sec CNT100;
   1:  PR[GP1:91,1] = PR[GP1:90,1] + -44.739;
   1:  PR[GP1:91,2] = PR[GP1:90,2] + -31.948;
   1:L PR[91] R[100]mm/sec CNT100;
   1:  PR[GP1:91,1] = PR[GP1:90,1] + -42.905;
   1:  PR[GP1:91,2] = PR[GP1:90,2] + -33.090;
   1:L PR[91] R[100]mm/sec CNT100;
   1:  PR[GP1:91,1] = PR[GP1:90,1] + -41.104;
   1:  PR[GP1:91,2] = PR[GP1:90,2] + -33.813;
   1:L PR[91] R[100]mm/sec CNT100;
   1:  PR[GP1:91,1] = PR[GP1:90,1] + -31.241;
   1:  PR[GP1:91,2] = PR[GP1:90,2] + -37.293;
   1:L PR[91] R[100]mm/sec CNT100;
   1:  PR[GP1:91,1] = PR[GP1:90,1] + -29.777;
   1:  PR[GP1:91,2] = PR[GP1:90,2] + -37.609;
   1:L PR[91] R[100]mm/sec CNT100;
   1:  PR[GP1:91,1] = PR[GP1:90,1] + -28.440;
   1:  PR[GP1:91,2] = PR[GP1:90,2] + -37.661;
   1:L PR[91] R[100]mm/sec CNT100;
   1:  PR[GP1:91,1] = PR[GP1:90,1] + -16.651;
   1:  PR[GP1:91,2] = PR[GP1:90,2] + -37.698;
   1:L PR[91] R[100]mm/sec CNT100;
   1:  PR[GP1:91,1] = PR[GP1:90,1] + -15.835;
   1:  PR[GP1:91,2] = PR[GP1:90,2] + -37.591;
   1:L PR[91] R[100]mm/sec CNT100;
   1:  PR[GP1:91,1] = PR[GP1:90,1] + -15.121;
   1:  PR[GP1:91,2] = PR[GP1:90,2] + -37.364;
   1:L PR[91] R[100]mm/sec CNT100;
   1:  PR[GP1:91,1] = PR[GP1:90,1] + -3.083;
   1:  PR[GP1:91,2] = PR[GP1:90,2] + -33.181;
   1:L PR[91] R[100]mm/sec CNT100;
   1:  PR[GP1:91,1] = PR[GP1:90,1] + -2.905;
   1:  PR[GP1:91,2] = PR[GP1:90,2] + -33.087;
   1:L PR[91] R[100]mm/sec CNT100;
   1:  PR[GP1:91,1] = PR[GP1:90,1] + -2.435;
   1:  PR[GP1:91,2] = PR[GP1:90,2] + -32.746;
   1:L PR[91] R[100]mm/sec CNT100;
   1:  PR[GP1:91,1] = PR[GP1:90,1] + 0.583;
   1:  PR[GP1:91,2] = PR[GP1:90,2] + -32.626;
   1:L PR[91] R[100]mm/sec CNT100;
   1:  PR[GP1:91,1] = PR[GP1:90,1] + 2.058;
   1:  PR[GP1:91,2] = PR[GP1:90,2] + -32.311;
   1:L PR[91] R[100]mm/sec CNT100;
   1:  PR[GP1:91,1] = PR[GP1:90,1] + 2.610;
   1:  PR[GP1:91,2] = PR[GP1:90,2] + -32.755;
   1:L PR[91] R[100]mm/sec CNT100;
   1:  PR[GP1:91,1] = PR[GP1:90,1] + 2.747;
   1:  PR[GP1:91,2] = PR[GP1:90,2] + -32.823;
   1:L PR[91] R[100]mm/sec CNT100;
   1:  PR[GP1:91,1] = PR[GP1:90,1] + 3.110;
   1:  PR[GP1:91,2] = PR[GP1:90,2] + -33.087;
   1:L PR[91] R[100]mm/sec CNT100;
   1:  PR[GP1:91,1] = PR[GP1:90,1] + 3.287;
   1:  PR[GP1:91,2] = PR[GP1:90,2] + -33.179;
   1:L PR[91] R[100]mm/sec CNT100;
   1:  PR[GP1:91,1] = PR[GP1:90,1] + 16.052;
   1:  PR[GP1:91,2] = PR[GP1:90,2] + -37.591;
   1:L PR[91] R[100]mm/sec CNT100;
   1:  PR[GP1:91,1] = PR[GP1:90,1] + 16.850;
   1:  PR[GP1:91,2] = PR[GP1:90,2] + -37.696;
   1:L PR[91] R[100]mm/sec CNT100;
   1:  PR[GP1:91,1] = PR[GP1:90,1] + 17.851;
   1:  PR[GP1:91,2] = PR[GP1:90,2] + -37.662;
   1:L PR[91] R[100]mm/sec CNT100;
   1:  PR[GP1:91,1] = PR[GP1:90,1] + 29.989;
   1:  PR[GP1:91,2] = PR[GP1:90,2] + -37.609;
   1:L PR[91] R[100]mm/sec CNT100;
   1:  PR[GP1:91,1] = PR[GP1:90,1] + 31.429;
   1:  PR[GP1:91,2] = PR[GP1:90,2] + -37.299;
   1:L PR[91] R[100]mm/sec CNT100;
   1:  PR[GP1:91,1] = PR[GP1:90,1] + 33.069;
   1:  PR[GP1:91,2] = PR[GP1:90,2] + -36.653;
   1:L PR[91] R[100]mm/sec CNT100;
   1:  PR[GP1:91,1] = PR[GP1:90,1] + 43.117;
   1:  PR[GP1:91,2] = PR[GP1:90,2] + -33.092;
   1:L PR[91] R[100]mm/sec CNT100;
   1:  PR[GP1:91,1] = PR[GP1:90,1] + 44.917;
   1:  PR[GP1:91,2] = PR[GP1:90,2] + -31.976;
   1:L PR[91] R[100]mm/sec CNT100;
   1:  PR[GP1:91,1] = PR[GP1:90,1] + 46.707;
   1:  PR[GP1:91,2] = PR[GP1:90,2] + -30.391;
   1:L PR[91] R[100]mm/sec CNT100;
   1:  PR[GP1:91,1] = PR[GP1:90,1] + 53.831;
   1:  PR[GP1:91,2] = PR[GP1:90,2] + -24.625;
   1:L PR[91] R[100]mm/sec CNT100;
   1:  PR[GP1:91,1] = PR[GP1:90,1] + 55.440;
   1:  PR[GP1:91,2] = PR[GP1:90,2] + -22.536;
   1:L PR[91] R[100]mm/sec CNT100;
   1:  PR[GP1:91,1] = PR[GP1:90,1] + 56.806;
   1:  PR[GP1:91,2] = PR[GP1:90,2] + -19.915;
   1:L PR[91] R[100]mm/sec CNT100;
   1:  PR[GP1:91,1] = PR[GP1:90,1] + 60.919;
   1:  PR[GP1:91,2] = PR[GP1:90,2] + -13.061;
   1:L PR[91] R[100]mm/sec CNT100;
   1:  PR[GP1:91,1] = PR[GP1:90,1] + 61.727;
   1:  PR[GP1:91,2] = PR[GP1:90,2] + -10.357;
   1:L PR[91] R[100]mm/sec CNT100;
   1:  PR[GP1:91,1] = PR[GP1:90,1] + 62.012;
   1:  PR[GP1:91,2] = PR[GP1:90,2] + -7.307;
   1:L PR[91] R[100]mm/sec CNT100;
   1:  PR[GP1:91,1] = PR[GP1:90,1] + 63.349;
   1:  PR[GP1:91,2] = PR[GP1:90,2] + -0.045;
   1:L PR[91] R[100]mm/sec CNT100;
   1:  PR[GP1:91,1] = PR[GP1:90,1] + 63.070;
   1:  PR[GP1:91,2] = PR[GP1:90,2] + 2.988;
   1:L PR[91] R[100]mm/sec CNT100;
   1:  PR[GP1:91,1] = PR[GP1:90,1] + 61.736;
   1:  PR[GP1:91,2] = PR[GP1:90,2] + 10.185;
   1:L PR[91] R[100]mm/sec CNT100;
   1:  PR[GP1:91,1] = PR[GP1:90,1] + 60.914;
   1:  PR[GP1:91,2] = PR[GP1:90,2] + 12.934;
   1:L PR[91] R[100]mm/sec CNT100;
   1:  PR[GP1:91,1] = PR[GP1:90,1] + 59.577;
   1:  PR[GP1:91,2] = PR[GP1:90,2] + 15.526;
   1:L PR[91] R[100]mm/sec CNT100;
   1:  PR[GP1:91,1] = PR[GP1:90,1] + 55.455;
   1:  PR[GP1:91,2] = PR[GP1:90,2] + 22.373;
   1:L PR[91] R[100]mm/sec CNT100;
   1:  PR[GP1:91,1] = PR[GP1:90,1] + 53.825;
   1:  PR[GP1:91,2] = PR[GP1:90,2] + 24.489;
   1:L PR[91] R[100]mm/sec CNT100;
   1:  PR[GP1:91,1] = PR[GP1:90,1] + 52.019;
   1:  PR[GP1:91,2] = PR[GP1:90,2] + 26.104;
   1:L PR[91] R[100]mm/sec CNT100;
   1:  PR[GP1:91,1] = PR[GP1:90,1] + 44.937;
   1:  PR[GP1:91,2] = PR[GP1:90,2] + 31.820;
   1:L PR[91] R[100]mm/sec CNT100;
   1:  PR[GP1:91,1] = PR[GP1:90,1] + 43.115;
   1:  PR[GP1:91,2] = PR[GP1:90,2] + 32.950;
   1:L PR[91] R[100]mm/sec CNT100;
   1:  PR[GP1:91,1] = PR[GP1:90,1] + 41.311;
   1:  PR[GP1:91,2] = PR[GP1:90,2] + 33.670;
   1:L PR[91] R[100]mm/sec CNT100;
   1:  PR[GP1:91,1] = PR[GP1:90,1] + 31.454;
   1:  PR[GP1:91,2] = PR[GP1:90,2] + 37.150;
   1:L PR[91] R[100]mm/sec CNT100;
   1:  PR[GP1:91,1] = PR[GP1:90,1] + 29.993;
   1:  PR[GP1:91,2] = PR[GP1:90,2] + 37.465;
   1:L PR[91] R[100]mm/sec CNT100;
   1:  PR[GP1:91,1] = PR[GP1:90,1] + 28.662;
   1:  PR[GP1:91,2] = PR[GP1:90,2] + 37.515;
   1:L PR[91] R[100]mm/sec CNT100;
   1:  PR[GP1:91,1] = PR[GP1:90,1] + 16.879;
   1:  PR[GP1:91,2] = PR[GP1:90,2] + 37.556;
   1:L PR[91] R[100]mm/sec CNT100;
   1:  PR[GP1:91,1] = PR[GP1:90,1] + 16.064;
   1:  PR[GP1:91,2] = PR[GP1:90,2] + 37.449;
   1:L PR[91] R[100]mm/sec CNT100;
   1:  PR[GP1:91,1] = PR[GP1:90,1] + 15.348;
   1:  PR[GP1:91,2] = PR[GP1:90,2] + 37.221;
   1:L PR[91] R[100]mm/sec CNT100;
   1:  PR[GP1:91,1] = PR[GP1:90,1] + 3.307;
   1:  PR[GP1:91,2] = PR[GP1:90,2] + 33.047;
   1:L PR[91] R[100]mm/sec CNT100;
   1:  PR[GP1:91,1] = PR[GP1:90,1] + 3.118;
   1:  PR[GP1:91,2] = PR[GP1:90,2] + 32.948;
   1:L PR[91] R[100]mm/sec CNT100;
   1:  PR[GP1:91,1] = PR[GP1:90,1] + 3.051;
   1:  PR[GP1:91,2] = PR[GP1:90,2] + 32.900;
   1:L PR[91] R[100]mm/sec CNT100;
   1:  PR[GP1:91,1] = PR[GP1:90,1] + 3.058;
   1:  PR[GP1:91,2] = PR[GP1:90,2] + 32.766;
   1:L PR[91] R[100]mm/sec CNT100;
   1:  PR[GP1:91,1] = PR[GP1:90,1] + 2.030;
   1:  PR[GP1:91,2] = PR[GP1:90,2] + 32.194;
   1:L PR[91] R[100]mm/sec CNT100;
   1:  ! -- Layer/Ebene 112 -- !;
   1:  PR[91] = PR[90];
   1:  PR[GP1:91,1] = PR[GP1:90,1] + -2.111;
   1:  PR[GP1:91,2] = PR[GP1:90,2] + 32.780;
   1:  PR[GP1:91,3] = PR[GP1:90,3] + 68.625;
   1:L PR[91] R[100]mm/sec CNT100;
   1:  PR[GP1:91,1] = PR[GP1:90,1] + -2.451;
   1:  PR[GP1:91,2] = PR[GP1:90,2] + 32.859;
   1:L PR[91] R[100]mm/sec CNT100;
   1:  PR[GP1:91,1] = PR[GP1:90,1] + -2.702;
   1:  PR[GP1:91,2] = PR[GP1:90,2] + 33.036;
   1:L PR[91] R[100]mm/sec CNT100;
   1:  PR[GP1:91,1] = PR[GP1:90,1] + -2.761;
   1:  PR[GP1:91,2] = PR[GP1:90,2] + 33.067;
   1:L PR[91] R[100]mm/sec CNT100;
   1:  PR[GP1:91,1] = PR[GP1:90,1] + -15.664;
   1:  PR[GP1:91,2] = PR[GP1:90,2] + 37.524;
   1:L PR[91] R[100]mm/sec CNT100;
   1:  PR[GP1:91,1] = PR[GP1:90,1] + -16.310;
   1:  PR[GP1:91,2] = PR[GP1:90,2] + 37.608;
   1:L PR[91] R[100]mm/sec CNT100;
   1:  PR[GP1:91,1] = PR[GP1:90,1] + -17.141;
   1:  PR[GP1:91,2] = PR[GP1:90,2] + 37.580;
   1:L PR[91] R[100]mm/sec CNT100;
   1:  PR[GP1:91,1] = PR[GP1:90,1] + -29.613;
   1:  PR[GP1:91,2] = PR[GP1:90,2] + 37.517;
   1:L PR[91] R[100]mm/sec CNT100;
   1:  PR[GP1:91,1] = PR[GP1:90,1] + -30.898;
   1:  PR[GP1:91,2] = PR[GP1:90,2] + 37.240;
   1:L PR[91] R[100]mm/sec CNT100;
   1:  PR[GP1:91,1] = PR[GP1:90,1] + -32.366;
   1:  PR[GP1:91,2] = PR[GP1:90,2] + 36.659;
   1:L PR[91] R[100]mm/sec CNT100;
   1:  PR[GP1:91,1] = PR[GP1:90,1] + -42.740;
   1:  PR[GP1:91,2] = PR[GP1:90,2] + 32.975;
   1:L PR[91] R[100]mm/sec CNT100;
   1:  PR[GP1:91,1] = PR[GP1:90,1] + -44.410;
   1:  PR[GP1:91,2] = PR[GP1:90,2] + 31.935;
   1:L PR[91] R[100]mm/sec CNT100;
   1:  PR[GP1:91,1] = PR[GP1:90,1] + -46.076;
   1:  PR[GP1:91,2] = PR[GP1:90,2] + 30.456;
   1:L PR[91] R[100]mm/sec CNT100;
   1:  PR[GP1:91,1] = PR[GP1:90,1] + -53.471;
   1:  PR[GP1:91,2] = PR[GP1:90,2] + 24.471;
   1:L PR[91] R[100]mm/sec CNT100;
   1:  PR[GP1:91,1] = PR[GP1:90,1] + -54.962;
   1:  PR[GP1:91,2] = PR[GP1:90,2] + 22.531;
   1:L PR[91] R[100]mm/sec CNT100;
   1:  PR[GP1:91,1] = PR[GP1:90,1] + -56.240;
   1:  PR[GP1:91,2] = PR[GP1:90,2] + 20.050;
   1:L PR[91] R[100]mm/sec CNT100;
   1:  PR[GP1:91,1] = PR[GP1:90,1] + -60.532;
   1:  PR[GP1:91,2] = PR[GP1:90,2] + 12.882;
   1:L PR[91] R[100]mm/sec CNT100;
   1:  PR[GP1:91,1] = PR[GP1:90,1] + -61.295;
   1:  PR[GP1:91,2] = PR[GP1:90,2] + 10.292;
   1:L PR[91] R[100]mm/sec CNT100;
   1:  PR[GP1:91,1] = PR[GP1:90,1] + -61.552;
   1:  PR[GP1:91,2] = PR[GP1:90,2] + 7.486;
   1:L PR[91] R[100]mm/sec CNT100;
   1:  PR[GP1:91,1] = PR[GP1:90,1] + -62.950;
   1:  PR[GP1:91,2] = PR[GP1:90,2] + -0.100;
   1:L PR[91] R[100]mm/sec CNT100;
   1:  PR[GP1:91,1] = PR[GP1:90,1] + -62.698;
   1:  PR[GP1:91,2] = PR[GP1:90,2] + -2.893;
   1:L PR[91] R[100]mm/sec CNT100;
   1:  PR[GP1:91,1] = PR[GP1:90,1] + -61.302;
   1:  PR[GP1:91,2] = PR[GP1:90,2] + -10.411;
   1:L PR[91] R[100]mm/sec CNT100;
   1:  PR[GP1:91,1] = PR[GP1:90,1] + -60.525;
   1:  PR[GP1:91,2] = PR[GP1:90,2] + -13.048;
   1:L PR[91] R[100]mm/sec CNT100;
   1:  PR[GP1:91,1] = PR[GP1:90,1] + -59.266;
   1:  PR[GP1:91,2] = PR[GP1:90,2] + -15.516;
   1:L PR[91] R[100]mm/sec CNT100;
   1:  PR[GP1:91,1] = PR[GP1:90,1] + -54.970;
   1:  PR[GP1:91,2] = PR[GP1:90,2] + -22.663;
   1:L PR[91] R[100]mm/sec CNT100;
   1:  PR[GP1:91,1] = PR[GP1:90,1] + -53.458;
   1:  PR[GP1:91,2] = PR[GP1:90,2] + -24.632;
   1:L PR[91] R[100]mm/sec CNT100;
   1:  PR[GP1:91,1] = PR[GP1:90,1] + -51.755;
   1:  PR[GP1:91,2] = PR[GP1:90,2] + -26.159;
   1:L PR[91] R[100]mm/sec CNT100;
   1:  PR[GP1:91,1] = PR[GP1:90,1] + -44.414;
   1:  PR[GP1:91,2] = PR[GP1:90,2] + -32.076;
   1:L PR[91] R[100]mm/sec CNT100;
   1:  PR[GP1:91,1] = PR[GP1:90,1] + -42.721;
   1:  PR[GP1:91,2] = PR[GP1:90,2] + -33.131;
   1:L PR[91] R[100]mm/sec CNT100;
   1:  PR[GP1:91,1] = PR[GP1:90,1] + -41.058;
   1:  PR[GP1:91,2] = PR[GP1:90,2] + -33.798;
   1:L PR[91] R[100]mm/sec CNT100;
   1:  PR[GP1:91,1] = PR[GP1:90,1] + -30.895;
   1:  PR[GP1:91,2] = PR[GP1:90,2] + -37.384;
   1:L PR[91] R[100]mm/sec CNT100;
   1:  PR[GP1:91,1] = PR[GP1:90,1] + -29.589;
   1:  PR[GP1:91,2] = PR[GP1:90,2] + -37.666;
   1:L PR[91] R[100]mm/sec CNT100;
   1:  PR[GP1:91,1] = PR[GP1:90,1] + -28.394;
   1:  PR[GP1:91,2] = PR[GP1:90,2] + -37.712;
   1:L PR[91] R[100]mm/sec CNT100;
   1:  PR[GP1:91,1] = PR[GP1:90,1] + -16.299;
   1:  PR[GP1:91,2] = PR[GP1:90,2] + -37.750;
   1:L PR[91] R[100]mm/sec CNT100;
   1:  PR[GP1:91,1] = PR[GP1:90,1] + -15.637;
   1:  PR[GP1:91,2] = PR[GP1:90,2] + -37.664;
   1:L PR[91] R[100]mm/sec CNT100;
   1:  PR[GP1:91,1] = PR[GP1:90,1] + -15.052;
   1:  PR[GP1:91,2] = PR[GP1:90,2] + -37.478;
   1:L PR[91] R[100]mm/sec CNT100;
   1:  PR[GP1:91,1] = PR[GP1:90,1] + -2.741;
   1:  PR[GP1:91,2] = PR[GP1:90,2] + -33.199;
   1:L PR[91] R[100]mm/sec CNT100;
   1:  PR[GP1:91,1] = PR[GP1:90,1] + -2.694;
   1:  PR[GP1:91,2] = PR[GP1:90,2] + -33.174;
   1:L PR[91] R[100]mm/sec CNT100;
   1:  PR[GP1:91,1] = PR[GP1:90,1] + -2.407;
   1:  PR[GP1:91,2] = PR[GP1:90,2] + -32.966;
   1:L PR[91] R[100]mm/sec CNT100;
   1:  PR[GP1:91,1] = PR[GP1:90,1] + 0.749;
   1:  PR[GP1:91,2] = PR[GP1:90,2] + -32.840;
   1:L PR[91] R[100]mm/sec CNT100;
   1:  PR[GP1:91,1] = PR[GP1:90,1] + 2.089;
   1:  PR[GP1:91,2] = PR[GP1:90,2] + -32.554;
   1:L PR[91] R[100]mm/sec CNT100;
   1:  PR[GP1:91,1] = PR[GP1:90,1] + 2.680;
   1:  PR[GP1:91,2] = PR[GP1:90,2] + -33.030;
   1:L PR[91] R[100]mm/sec CNT100;
   1:  PR[GP1:91,1] = PR[GP1:90,1] + 2.964;
   1:  PR[GP1:91,2] = PR[GP1:90,2] + -33.204;
   1:L PR[91] R[100]mm/sec CNT100;
   1:  PR[GP1:91,1] = PR[GP1:90,1] + 15.854;
   1:  PR[GP1:91,2] = PR[GP1:90,2] + -37.663;
   1:L PR[91] R[100]mm/sec CNT100;
   1:  PR[GP1:91,1] = PR[GP1:90,1] + 16.498;
   1:  PR[GP1:91,2] = PR[GP1:90,2] + -37.748;
   1:L PR[91] R[100]mm/sec CNT100;
   1:  PR[GP1:91,1] = PR[GP1:90,1] + 17.324;
   1:  PR[GP1:91,2] = PR[GP1:90,2] + -37.720;
   1:L PR[91] R[100]mm/sec CNT100;
   1:  PR[GP1:91,1] = PR[GP1:90,1] + 29.802;
   1:  PR[GP1:91,2] = PR[GP1:90,2] + -37.665;
   1:L PR[91] R[100]mm/sec CNT100;
   1:  PR[GP1:91,1] = PR[GP1:90,1] + 31.084;
   1:  PR[GP1:91,2] = PR[GP1:90,2] + -37.389;
   1:L PR[91] R[100]mm/sec CNT100;
   1:  PR[GP1:91,1] = PR[GP1:90,1] + 32.553;
   1:  PR[GP1:91,2] = PR[GP1:90,2] + -36.811;
   1:L PR[91] R[100]mm/sec CNT100;
   1:  PR[GP1:91,1] = PR[GP1:90,1] + 42.934;
   1:  PR[GP1:91,2] = PR[GP1:90,2] + -33.132;
   1:L PR[91] R[100]mm/sec CNT100;
   1:  PR[GP1:91,1] = PR[GP1:90,1] + 44.594;
   1:  PR[GP1:91,2] = PR[GP1:90,2] + -32.103;
   1:L PR[91] R[100]mm/sec CNT100;
   1:  PR[GP1:91,1] = PR[GP1:90,1] + 46.249;
   1:  PR[GP1:91,2] = PR[GP1:90,2] + -30.637;
   1:L PR[91] R[100]mm/sec CNT100;
   1:  PR[GP1:91,1] = PR[GP1:90,1] + 53.649;
   1:  PR[GP1:91,2] = PR[GP1:90,2] + -24.647;
   1:L PR[91] R[100]mm/sec CNT100;
   1:  PR[GP1:91,1] = PR[GP1:90,1] + 55.156;
   1:  PR[GP1:91,2] = PR[GP1:90,2] + -22.691;
   1:L PR[91] R[100]mm/sec CNT100;
   1:  PR[GP1:91,1] = PR[GP1:90,1] + 56.438;
   1:  PR[GP1:91,2] = PR[GP1:90,2] + -20.230;
   1:L PR[91] R[100]mm/sec CNT100;
   1:  PR[GP1:91,1] = PR[GP1:90,1] + 60.733;
   1:  PR[GP1:91,2] = PR[GP1:90,2] + -13.075;
   1:L PR[91] R[100]mm/sec CNT100;
   1:  PR[GP1:91,1] = PR[GP1:90,1] + 61.495;
   1:  PR[GP1:91,2] = PR[GP1:90,2] + -10.525;
   1:L PR[91] R[100]mm/sec CNT100;
   1:  PR[GP1:91,1] = PR[GP1:90,1] + 61.764;
   1:  PR[GP1:91,2] = PR[GP1:90,2] + -7.642;
   1:L PR[91] R[100]mm/sec CNT100;
   1:  PR[GP1:91,1] = PR[GP1:90,1] + 63.163;
   1:  PR[GP1:91,2] = PR[GP1:90,2] + -0.045;
   1:L PR[91] R[100]mm/sec CNT100;
   1:  PR[GP1:91,1] = PR[GP1:90,1] + 62.898;
   1:  PR[GP1:91,2] = PR[GP1:90,2] + 2.827;
   1:L PR[91] R[100]mm/sec CNT100;
   1:  PR[GP1:91,1] = PR[GP1:90,1] + 61.503;
   1:  PR[GP1:91,2] = PR[GP1:90,2] + 10.353;
   1:L PR[91] R[100]mm/sec CNT100;
   1:  PR[GP1:91,1] = PR[GP1:90,1] + 60.728;
   1:  PR[GP1:91,2] = PR[GP1:90,2] + 12.948;
   1:L PR[91] R[100]mm/sec CNT100;
   1:  PR[GP1:91,1] = PR[GP1:90,1] + 59.465;
   1:  PR[GP1:91,2] = PR[GP1:90,2] + 15.395;
   1:L PR[91] R[100]mm/sec CNT100;
   1:  PR[GP1:91,1] = PR[GP1:90,1] + 55.171;
   1:  PR[GP1:91,2] = PR[GP1:90,2] + 22.528;
   1:L PR[91] R[100]mm/sec CNT100;
   1:  PR[GP1:91,1] = PR[GP1:90,1] + 53.644;
   1:  PR[GP1:91,2] = PR[GP1:90,2] + 24.511;
   1:L PR[91] R[100]mm/sec CNT100;
   1:  PR[GP1:91,1] = PR[GP1:90,1] + 51.950;
   1:  PR[GP1:91,2] = PR[GP1:90,2] + 26.025;
   1:L PR[91] R[100]mm/sec CNT100;
   1:  PR[GP1:91,1] = PR[GP1:90,1] + 44.614;
   1:  PR[GP1:91,2] = PR[GP1:90,2] + 31.947;
   1:L PR[91] R[100]mm/sec CNT100;
   1:  PR[GP1:91,1] = PR[GP1:90,1] + 42.932;
   1:  PR[GP1:91,2] = PR[GP1:90,2] + 32.989;
   1:L PR[91] R[100]mm/sec CNT100;
   1:  PR[GP1:91,1] = PR[GP1:90,1] + 41.267;
   1:  PR[GP1:91,2] = PR[GP1:90,2] + 33.655;
   1:L PR[91] R[100]mm/sec CNT100;
   1:  PR[GP1:91,1] = PR[GP1:90,1] + 31.109;
   1:  PR[GP1:91,2] = PR[GP1:90,2] + 37.241;
   1:L PR[91] R[100]mm/sec CNT100;
   1:  PR[GP1:91,1] = PR[GP1:90,1] + 29.806;
   1:  PR[GP1:91,2] = PR[GP1:90,2] + 37.521;
   1:L PR[91] R[100]mm/sec CNT100;
   1:  PR[GP1:91,1] = PR[GP1:90,1] + 28.617;
   1:  PR[GP1:91,2] = PR[GP1:90,2] + 37.566;
   1:L PR[91] R[100]mm/sec CNT100;
   1:  PR[GP1:91,1] = PR[GP1:90,1] + 16.527;
   1:  PR[GP1:91,2] = PR[GP1:90,2] + 37.608;
   1:L PR[91] R[100]mm/sec CNT100;
   1:  PR[GP1:91,1] = PR[GP1:90,1] + 15.866;
   1:  PR[GP1:91,2] = PR[GP1:90,2] + 37.521;
   1:L PR[91] R[100]mm/sec CNT100;
   1:  PR[GP1:91,1] = PR[GP1:90,1] + 15.280;
   1:  PR[GP1:91,2] = PR[GP1:90,2] + 37.335;
   1:L PR[91] R[100]mm/sec CNT100;
   1:  PR[GP1:91,1] = PR[GP1:90,1] + 3.024;
   1:  PR[GP1:91,2] = PR[GP1:90,2] + 33.086;
   1:L PR[91] R[100]mm/sec CNT100;
   1:  PR[GP1:91,1] = PR[GP1:90,1] + 3.030;
   1:  PR[GP1:91,2] = PR[GP1:90,2] + 32.977;
   1:L PR[91] R[100]mm/sec CNT100;
   1:  PR[GP1:91,1] = PR[GP1:90,1] + 2.060;
   1:  PR[GP1:91,2] = PR[GP1:90,2] + 32.437;
   1:L PR[91] R[100]mm/sec CNT100;
   1:  ! -- Layer/Ebene 113 -- !;
   1:  PR[91] = PR[90];
   1:  PR[GP1:91,1] = PR[GP1:90,1] + -2.298;
   1:  PR[GP1:91,2] = PR[GP1:90,2] + 33.042;
   1:  PR[GP1:91,3] = PR[GP1:90,3] + 69.235;
   1:L PR[91] R[100]mm/sec CNT100;
   1:  PR[GP1:91,1] = PR[GP1:90,1] + -15.466;
   1:  PR[GP1:91,2] = PR[GP1:90,2] + 37.596;
   1:L PR[91] R[100]mm/sec CNT100;
   1:  PR[GP1:91,1] = PR[GP1:90,1] + -15.959;
   1:  PR[GP1:91,2] = PR[GP1:90,2] + 37.660;
   1:L PR[91] R[100]mm/sec CNT100;
   1:  PR[GP1:91,1] = PR[GP1:90,1] + -16.613;
   1:  PR[GP1:91,2] = PR[GP1:90,2] + 37.638;
   1:L PR[91] R[100]mm/sec CNT100;
   1:  PR[GP1:91,1] = PR[GP1:90,1] + -29.426;
   1:  PR[GP1:91,2] = PR[GP1:90,2] + 37.574;
   1:L PR[91] R[100]mm/sec CNT100;
   1:  PR[GP1:91,1] = PR[GP1:90,1] + -30.553;
   1:  PR[GP1:91,2] = PR[GP1:90,2] + 37.331;
   1:L PR[91] R[100]mm/sec CNT100;
   1:  PR[GP1:91,1] = PR[GP1:90,1] + -31.850;
   1:  PR[GP1:91,2] = PR[GP1:90,2] + 36.817;
   1:L PR[91] R[100]mm/sec CNT100;
   1:  PR[GP1:91,1] = PR[GP1:90,1] + -42.556;
   1:  PR[GP1:91,2] = PR[GP1:90,2] + 33.015;
   1:L PR[91] R[100]mm/sec CNT100;
   1:  PR[GP1:91,1] = PR[GP1:90,1] + -44.085;
   1:  PR[GP1:91,2] = PR[GP1:90,2] + 32.063;
   1:L PR[91] R[100]mm/sec CNT100;
   1:  PR[GP1:91,1] = PR[GP1:90,1] + -45.615;
   1:  PR[GP1:91,2] = PR[GP1:90,2] + 30.704;
   1:L PR[91] R[100]mm/sec CNT100;
   1:  PR[GP1:91,1] = PR[GP1:90,1] + -53.288;
   1:  PR[GP1:91,2] = PR[GP1:90,2] + 24.495;
   1:L PR[91] R[100]mm/sec CNT100;
   1:  PR[GP1:91,1] = PR[GP1:90,1] + -54.677;
   1:  PR[GP1:91,2] = PR[GP1:90,2] + 22.687;
   1:L PR[91] R[100]mm/sec CNT100;
   1:  PR[GP1:91,1] = PR[GP1:90,1] + -55.872;
   1:  PR[GP1:91,2] = PR[GP1:90,2] + 20.368;
   1:L PR[91] R[100]mm/sec CNT100;
   1:  PR[GP1:91,1] = PR[GP1:90,1] + -60.345;
   1:  PR[GP1:91,2] = PR[GP1:90,2] + 12.897;
   1:L PR[91] R[100]mm/sec CNT100;
   1:  PR[GP1:91,1] = PR[GP1:90,1] + -61.062;
   1:  PR[GP1:91,2] = PR[GP1:90,2] + 10.463;
   1:L PR[91] R[100]mm/sec CNT100;
   1:  PR[GP1:91,1] = PR[GP1:90,1] + -61.304;
   1:  PR[GP1:91,2] = PR[GP1:90,2] + 7.820;
   1:L PR[91] R[100]mm/sec CNT100;
   1:  PR[GP1:91,1] = PR[GP1:90,1] + -62.764;
   1:  PR[GP1:91,2] = PR[GP1:90,2] + -0.100;
   1:L PR[91] R[100]mm/sec CNT100;
   1:  PR[GP1:91,1] = PR[GP1:90,1] + -62.526;
   1:  PR[GP1:91,2] = PR[GP1:90,2] + -2.736;
   1:L PR[91] R[100]mm/sec CNT100;
   1:  PR[GP1:91,1] = PR[GP1:90,1] + -61.069;
   1:  PR[GP1:91,2] = PR[GP1:90,2] + -10.583;
   1:L PR[91] R[100]mm/sec CNT100;
   1:  PR[GP1:91,1] = PR[GP1:90,1] + -60.338;
   1:  PR[GP1:91,2] = PR[GP1:90,2] + -13.063;
   1:L PR[91] R[100]mm/sec CNT100;
   1:  PR[GP1:91,1] = PR[GP1:90,1] + -59.153;
   1:  PR[GP1:91,2] = PR[GP1:90,2] + -15.386;
   1:L PR[91] R[100]mm/sec CNT100;
   1:  PR[GP1:91,1] = PR[GP1:90,1] + -54.685;
   1:  PR[GP1:91,2] = PR[GP1:90,2] + -22.820;
   1:L PR[91] R[100]mm/sec CNT100;
   1:  PR[GP1:91,1] = PR[GP1:90,1] + -53.274;
   1:  PR[GP1:91,2] = PR[GP1:90,2] + -24.656;
   1:L PR[91] R[100]mm/sec CNT100;
   1:  PR[GP1:91,1] = PR[GP1:90,1] + -51.685;
   1:  PR[GP1:91,2] = PR[GP1:90,2] + -26.082;
   1:L PR[91] R[100]mm/sec CNT100;
   1:  PR[GP1:91,1] = PR[GP1:90,1] + -44.089;
   1:  PR[GP1:91,2] = PR[GP1:90,2] + -32.204;
   1:L PR[91] R[100]mm/sec CNT100;
   1:  PR[GP1:91,1] = PR[GP1:90,1] + -42.537;
   1:  PR[GP1:91,2] = PR[GP1:90,2] + -33.171;
   1:L PR[91] R[100]mm/sec CNT100;
   1:  PR[GP1:91,1] = PR[GP1:90,1] + -41.012;
   1:  PR[GP1:91,2] = PR[GP1:90,2] + -33.783;
   1:L PR[91] R[100]mm/sec CNT100;
   1:  PR[GP1:91,1] = PR[GP1:90,1] + -30.549;
   1:  PR[GP1:91,2] = PR[GP1:90,2] + -37.475;
   1:L PR[91] R[100]mm/sec CNT100;
   1:  PR[GP1:91,1] = PR[GP1:90,1] + -29.401;
   1:  PR[GP1:91,2] = PR[GP1:90,2] + -37.722;
   1:L PR[91] R[100]mm/sec CNT100;
   1:  PR[GP1:91,1] = PR[GP1:90,1] + -28.349;
   1:  PR[GP1:91,2] = PR[GP1:90,2] + -37.763;
   1:L PR[91] R[100]mm/sec CNT100;
   1:  PR[GP1:91,1] = PR[GP1:90,1] + -15.947;
   1:  PR[GP1:91,2] = PR[GP1:90,2] + -37.802;
   1:L PR[91] R[100]mm/sec CNT100;
   1:  PR[GP1:91,1] = PR[GP1:90,1] + -15.438;
   1:  PR[GP1:91,2] = PR[GP1:90,2] + -37.736;
   1:L PR[91] R[100]mm/sec CNT100;
   1:  PR[GP1:91,1] = PR[GP1:90,1] + -14.984;
   1:  PR[GP1:91,2] = PR[GP1:90,2] + -37.591;
   1:L PR[91] R[100]mm/sec CNT100;
   1:  PR[GP1:91,1] = PR[GP1:90,1] + -2.286;
   1:  PR[GP1:91,2] = PR[GP1:90,2] + -33.182;
   1:L PR[91] R[100]mm/sec CNT100;
   1:  PR[GP1:91,1] = PR[GP1:90,1] + 0.914;
   1:  PR[GP1:91,2] = PR[GP1:90,2] + -33.055;
   1:L PR[91] R[100]mm/sec CNT100;
   1:  PR[GP1:91,1] = PR[GP1:90,1] + 2.119;
   1:  PR[GP1:91,2] = PR[GP1:90,2] + -32.798;
   1:L PR[91] R[100]mm/sec CNT100;
   1:  PR[GP1:91,1] = PR[GP1:90,1] + 2.673;
   1:  PR[GP1:91,2] = PR[GP1:90,2] + -33.244;
   1:L PR[91] R[100]mm/sec CNT100;
   1:  PR[GP1:91,1] = PR[GP1:90,1] + 15.655;
   1:  PR[GP1:91,2] = PR[GP1:90,2] + -37.735;
   1:L PR[91] R[100]mm/sec CNT100;
   1:  PR[GP1:91,1] = PR[GP1:90,1] + 16.146;
   1:  PR[GP1:91,2] = PR[GP1:90,2] + -37.800;
   1:L PR[91] R[100]mm/sec CNT100;
   1:  PR[GP1:91,1] = PR[GP1:90,1] + 16.796;
   1:  PR[GP1:91,2] = PR[GP1:90,2] + -37.778;
   1:L PR[91] R[100]mm/sec CNT100;
   1:  PR[GP1:91,1] = PR[GP1:90,1] + 29.615;
   1:  PR[GP1:91,2] = PR[GP1:90,2] + -37.722;
   1:L PR[91] R[100]mm/sec CNT100;
   1:  PR[GP1:91,1] = PR[GP1:90,1] + 30.739;
   1:  PR[GP1:91,2] = PR[GP1:90,2] + -37.480;
   1:L PR[91] R[100]mm/sec CNT100;
   1:  PR[GP1:91,1] = PR[GP1:90,1] + 32.038;
   1:  PR[GP1:91,2] = PR[GP1:90,2] + -36.968;
   1:L PR[91] R[100]mm/sec CNT100;
   1:  PR[GP1:91,1] = PR[GP1:90,1] + 42.751;
   1:  PR[GP1:91,2] = PR[GP1:90,2] + -33.172;
   1:L PR[91] R[100]mm/sec CNT100;
   1:  PR[GP1:91,1] = PR[GP1:90,1] + 44.270;
   1:  PR[GP1:91,2] = PR[GP1:90,2] + -32.230;
   1:L PR[91] R[100]mm/sec CNT100;
   1:  PR[GP1:91,1] = PR[GP1:90,1] + 45.791;
   1:  PR[GP1:91,2] = PR[GP1:90,2] + -30.883;
   1:L PR[91] R[100]mm/sec CNT100;
   1:  PR[GP1:91,1] = PR[GP1:90,1] + 53.468;
   1:  PR[GP1:91,2] = PR[GP1:90,2] + -24.669;
   1:L PR[91] R[100]mm/sec CNT100;
   1:  PR[GP1:91,1] = PR[GP1:90,1] + 54.872;
   1:  PR[GP1:91,2] = PR[GP1:90,2] + -22.845;
   1:L PR[91] R[100]mm/sec CNT100;
   1:  PR[GP1:91,1] = PR[GP1:90,1] + 56.071;
   1:  PR[GP1:91,2] = PR[GP1:90,2] + -20.546;
   1:L PR[91] R[100]mm/sec CNT100;
   1:  PR[GP1:91,1] = PR[GP1:90,1] + 60.546;
   1:  PR[GP1:91,2] = PR[GP1:90,2] + -13.089;
   1:L PR[91] R[100]mm/sec CNT100;
   1:  PR[GP1:91,1] = PR[GP1:90,1] + 61.262;
   1:  PR[GP1:91,2] = PR[GP1:90,2] + -10.693;
   1:L PR[91] R[100]mm/sec CNT100;
   1:  PR[GP1:91,1] = PR[GP1:90,1] + 61.516;
   1:  PR[GP1:91,2] = PR[GP1:90,2] + -7.977;
   1:L PR[91] R[100]mm/sec CNT100;
   1:  PR[GP1:91,1] = PR[GP1:90,1] + 62.977;
   1:  PR[GP1:91,2] = PR[GP1:90,2] + -0.045;
   1:L PR[91] R[100]mm/sec CNT100;
   1:  PR[GP1:91,1] = PR[GP1:90,1] + 62.727;
   1:  PR[GP1:91,2] = PR[GP1:90,2] + 2.667;
   1:L PR[91] R[100]mm/sec CNT100;
   1:  PR[GP1:91,1] = PR[GP1:90,1] + 61.271;
   1:  PR[GP1:91,2] = PR[GP1:90,2] + 10.520;
   1:L PR[91] R[100]mm/sec CNT100;
   1:  PR[GP1:91,1] = PR[GP1:90,1] + 60.542;
   1:  PR[GP1:91,2] = PR[GP1:90,2] + 12.962;
   1:L PR[91] R[100]mm/sec CNT100;
   1:  PR[GP1:91,1] = PR[GP1:90,1] + 59.353;
   1:  PR[GP1:91,2] = PR[GP1:90,2] + 15.265;
   1:L PR[91] R[100]mm/sec CNT100;
   1:  PR[GP1:91,1] = PR[GP1:90,1] + 54.887;
   1:  PR[GP1:91,2] = PR[GP1:90,2] + 22.682;
   1:L PR[91] R[100]mm/sec CNT100;
   1:  PR[GP1:91,1] = PR[GP1:90,1] + 53.462;
   1:  PR[GP1:91,2] = PR[GP1:90,2] + 24.533;
   1:L PR[91] R[100]mm/sec CNT100;
   1:  PR[GP1:91,1] = PR[GP1:90,1] + 51.881;
   1:  PR[GP1:91,2] = PR[GP1:90,2] + 25.946;
   1:L PR[91] R[100]mm/sec CNT100;
   1:  PR[GP1:91,1] = PR[GP1:90,1] + 44.290;
   1:  PR[GP1:91,2] = PR[GP1:90,2] + 32.074;
   1:L PR[91] R[100]mm/sec CNT100;
   1:  PR[GP1:91,1] = PR[GP1:90,1] + 42.749;
   1:  PR[GP1:91,2] = PR[GP1:90,2] + 33.029;
   1:L PR[91] R[100]mm/sec CNT100;
   1:  PR[GP1:91,1] = PR[GP1:90,1] + 41.222;
   1:  PR[GP1:91,2] = PR[GP1:90,2] + 33.639;
   1:L PR[91] R[100]mm/sec CNT100;
   1:  PR[GP1:91,1] = PR[GP1:90,1] + 30.765;
   1:  PR[GP1:91,2] = PR[GP1:90,2] + 37.331;
   1:L PR[91] R[100]mm/sec CNT100;
   1:  PR[GP1:91,1] = PR[GP1:90,1] + 29.619;
   1:  PR[GP1:91,2] = PR[GP1:90,2] + 37.578;
   1:L PR[91] R[100]mm/sec CNT100;
   1:  PR[GP1:91,1] = PR[GP1:90,1] + 28.572;
   1:  PR[GP1:91,2] = PR[GP1:90,2] + 37.617;
   1:L PR[91] R[100]mm/sec CNT100;
   1:  PR[GP1:91,1] = PR[GP1:90,1] + 16.176;
   1:  PR[GP1:91,2] = PR[GP1:90,2] + 37.661;
   1:L PR[91] R[100]mm/sec CNT100;
   1:  PR[GP1:91,1] = PR[GP1:90,1] + 15.667;
   1:  PR[GP1:91,2] = PR[GP1:90,2] + 37.594;
   1:L PR[91] R[100]mm/sec CNT100;
   1:  PR[GP1:91,1] = PR[GP1:90,1] + 15.212;
   1:  PR[GP1:91,2] = PR[GP1:90,2] + 37.449;
   1:L PR[91] R[100]mm/sec CNT100;
   1:  PR[GP1:91,1] = PR[GP1:90,1] + 2.987;
   1:  PR[GP1:91,2] = PR[GP1:90,2] + 33.210;
   1:L PR[91] R[100]mm/sec CNT100;
   1:  PR[GP1:91,2] = PR[GP1:90,2] + 33.180;
   1:L PR[91] R[100]mm/sec CNT100;
   1:  PR[GP1:91,1] = PR[GP1:90,1] + 2.090;
   1:  PR[GP1:91,2] = PR[GP1:90,2] + 32.680;
   1:L PR[91] R[100]mm/sec CNT100;
   1:  ! -- Layer/Ebene 114 -- !;
   1:  PR[91] = PR[90];
   1:  PR[GP1:91,1] = PR[GP1:90,1] + -1.618;
   1:  PR[GP1:91,2] = PR[GP1:90,2] + 33.231;
   1:  PR[GP1:91,3] = PR[GP1:90,3] + 69.845;
   1:L PR[91] R[100]mm/sec CNT100;
   1:  PR[GP1:91,1] = PR[GP1:90,1] + -2.240;
   1:  PR[GP1:91,2] = PR[GP1:90,2] + 33.227;
   1:L PR[91] R[100]mm/sec CNT100;
   1:  PR[GP1:91,1] = PR[GP1:90,1] + -5.452;
   1:  PR[GP1:91,2] = PR[GP1:90,2] + 34.275;
   1:L PR[91] R[100]mm/sec CNT100;
   1:  PR[GP1:91,1] = PR[GP1:90,1] + -15.267;
   1:  PR[GP1:91,2] = PR[GP1:90,2] + 37.668;
   1:L PR[91] R[100]mm/sec CNT100;
   1:  PR[GP1:91,1] = PR[GP1:90,1] + -15.607;
   1:  PR[GP1:91,2] = PR[GP1:90,2] + 37.713;
   1:L PR[91] R[100]mm/sec CNT100;
   1:  PR[GP1:91,1] = PR[GP1:90,1] + -16.084;
   1:  PR[GP1:91,2] = PR[GP1:90,2] + 37.696;
   1:L PR[91] R[100]mm/sec CNT100;
   1:  PR[GP1:91,1] = PR[GP1:90,1] + -29.238;
   1:  PR[GP1:91,2] = PR[GP1:90,2] + 37.630;
   1:L PR[91] R[100]mm/sec CNT100;
   1:  PR[GP1:91,1] = PR[GP1:90,1] + -30.207;
   1:  PR[GP1:91,2] = PR[GP1:90,2] + 37.421;
   1:L PR[91] R[100]mm/sec CNT100;
   1:  PR[GP1:91,1] = PR[GP1:90,1] + -31.334;
   1:  PR[GP1:91,2] = PR[GP1:90,2] + 36.975;
   1:L PR[91] R[100]mm/sec CNT100;
   1:  PR[GP1:91,1] = PR[GP1:90,1] + -42.373;
   1:  PR[GP1:91,2] = PR[GP1:90,2] + 33.055;
   1:L PR[91] R[100]mm/sec CNT100;
   1:  PR[GP1:91,1] = PR[GP1:90,1] + -43.760;
   1:  PR[GP1:91,2] = PR[GP1:90,2] + 32.191;
   1:L PR[91] R[100]mm/sec CNT100;
   1:  PR[GP1:91,1] = PR[GP1:90,1] + -45.155;
   1:  PR[GP1:91,2] = PR[GP1:90,2] + 30.953;
   1:L PR[91] R[100]mm/sec CNT100;
   1:  PR[GP1:91,1] = PR[GP1:90,1] + -53.104;
   1:  PR[GP1:91,2] = PR[GP1:90,2] + 24.520;
   1:L PR[91] R[100]mm/sec CNT100;
   1:  PR[GP1:91,1] = PR[GP1:90,1] + -54.393;
   1:  PR[GP1:91,2] = PR[GP1:90,2] + 22.843;
   1:L PR[91] R[100]mm/sec CNT100;
   1:  PR[GP1:91,1] = PR[GP1:90,1] + -55.504;
   1:  PR[GP1:91,2] = PR[GP1:90,2] + 20.686;
   1:L PR[91] R[100]mm/sec CNT100;
   1:  PR[GP1:91,1] = PR[GP1:90,1] + -60.158;
   1:  PR[GP1:91,2] = PR[GP1:90,2] + 12.913;
   1:L PR[91] R[100]mm/sec CNT100;
   1:  PR[GP1:91,1] = PR[GP1:90,1] + -60.829;
   1:  PR[GP1:91,2] = PR[GP1:90,2] + 10.635;
   1:L PR[91] R[100]mm/sec CNT100;
   1:  PR[GP1:91,1] = PR[GP1:90,1] + -61.056;
   1:  PR[GP1:91,2] = PR[GP1:90,2] + 8.154;
   1:L PR[91] R[100]mm/sec CNT100;
   1:  PR[GP1:91,1] = PR[GP1:90,1] + -62.577;
   1:  PR[GP1:91,2] = PR[GP1:90,2] + -0.100;
   1:L PR[91] R[100]mm/sec CNT100;
   1:  PR[GP1:91,1] = PR[GP1:90,1] + -62.353;
   1:  PR[GP1:91,2] = PR[GP1:90,2] + -2.580;
   1:L PR[91] R[100]mm/sec CNT100;
   1:  PR[GP1:91,1] = PR[GP1:90,1] + -60.836;
   1:  PR[GP1:91,2] = PR[GP1:90,2] + -10.755;
   1:L PR[91] R[100]mm/sec CNT100;
   1:  PR[GP1:91,1] = PR[GP1:90,1] + -60.151;
   1:  PR[GP1:91,2] = PR[GP1:90,2] + -13.079;
   1:L PR[91] R[100]mm/sec CNT100;
   1:  PR[GP1:91,1] = PR[GP1:90,1] + -59.040;
   1:  PR[GP1:91,2] = PR[GP1:90,2] + -15.257;
   1:L PR[91] R[100]mm/sec CNT100;
   1:  PR[GP1:91,1] = PR[GP1:90,1] + -54.401;
   1:  PR[GP1:91,2] = PR[GP1:90,2] + -22.976;
   1:L PR[91] R[100]mm/sec CNT100;
   1:  PR[GP1:91,1] = PR[GP1:90,1] + -53.091;
   1:  PR[GP1:91,2] = PR[GP1:90,2] + -24.680;
   1:L PR[91] R[100]mm/sec CNT100;
   1:  PR[GP1:91,1] = PR[GP1:90,1] + -51.615;
   1:  PR[GP1:91,2] = PR[GP1:90,2] + -26.004;
   1:L PR[91] R[100]mm/sec CNT100;
   1:  PR[GP1:91,1] = PR[GP1:90,1] + -43.763;
   1:  PR[GP1:91,2] = PR[GP1:90,2] + -32.333;
   1:L PR[91] R[100]mm/sec CNT100;
   1:  PR[GP1:91,1] = PR[GP1:90,1] + -42.353;
   1:  PR[GP1:91,2] = PR[GP1:90,2] + -33.211;
   1:L PR[91] R[100]mm/sec CNT100;
   1:  PR[GP1:91,1] = PR[GP1:90,1] + -40.967;
   1:  PR[GP1:91,2] = PR[GP1:90,2] + -33.768;
   1:L PR[91] R[100]mm/sec CNT100;
   1:  PR[GP1:91,1] = PR[GP1:90,1] + -30.202;
   1:  PR[GP1:91,2] = PR[GP1:90,2] + -37.566;
   1:L PR[91] R[100]mm/sec CNT100;
   1:  PR[GP1:91,1] = PR[GP1:90,1] + -29.213;
   1:  PR[GP1:91,2] = PR[GP1:90,2] + -37.779;
   1:L PR[91] R[100]mm/sec CNT100;
   1:  PR[GP1:91,1] = PR[GP1:90,1] + -28.303;
   1:  PR[GP1:91,2] = PR[GP1:90,2] + -37.814;
   1:L PR[91] R[100]mm/sec CNT100;
   1:  PR[GP1:91,1] = PR[GP1:90,1] + -15.595;
   1:  PR[GP1:91,2] = PR[GP1:90,2] + -37.854;
   1:L PR[91] R[100]mm/sec CNT100;
   1:  PR[GP1:91,1] = PR[GP1:90,1] + -15.239;
   1:  PR[GP1:91,2] = PR[GP1:90,2] + -37.808;
   1:L PR[91] R[100]mm/sec CNT100;
   1:  PR[GP1:91,1] = PR[GP1:90,1] + -14.915;
   1:  PR[GP1:91,2] = PR[GP1:90,2] + -37.705;
   1:L PR[91] R[100]mm/sec CNT100;
   1:  PR[GP1:91,1] = PR[GP1:90,1] + -5.612;
   1:  PR[GP1:91,2] = PR[GP1:90,2] + -34.472;
   1:L PR[91] R[100]mm/sec CNT100;
   1:  PR[GP1:91,1] = PR[GP1:90,1] + -2.240;
   1:  PR[GP1:91,2] = PR[GP1:90,2] + -33.372;
   1:L PR[91] R[100]mm/sec CNT100;
   1:  PR[GP1:91,1] = PR[GP1:90,1] + -1.558;
   1:  PR[GP1:91,2] = PR[GP1:90,2] + -33.375;
   1:L PR[91] R[100]mm/sec CNT100;
   1:  PR[GP1:91,1] = PR[GP1:90,1] + 1.080;
   1:  PR[GP1:91,2] = PR[GP1:90,2] + -33.270;
   1:L PR[91] R[100]mm/sec CNT100;
   1:  PR[GP1:91,1] = PR[GP1:90,1] + 2.150;
   1:  PR[GP1:91,2] = PR[GP1:90,2] + -33.041;
   1:L PR[91] R[100]mm/sec CNT100;
   1:  PR[GP1:91,1] = PR[GP1:90,1] + 2.642;
   1:  PR[GP1:91,2] = PR[GP1:90,2] + -33.438;
   1:L PR[91] R[100]mm/sec CNT100;
   1:  PR[GP1:91,1] = PR[GP1:90,1] + 5.822;
   1:  PR[GP1:91,2] = PR[GP1:90,2] + -34.472;
   1:L PR[91] R[100]mm/sec CNT100;
   1:  PR[GP1:91,1] = PR[GP1:90,1] + 15.456;
   1:  PR[GP1:91,2] = PR[GP1:90,2] + -37.808;
   1:L PR[91] R[100]mm/sec CNT100;
   1:  PR[GP1:91,1] = PR[GP1:90,1] + 15.794;
   1:  PR[GP1:91,2] = PR[GP1:90,2] + -37.852;
   1:L PR[91] R[100]mm/sec CNT100;
   1:  PR[GP1:91,1] = PR[GP1:90,1] + 16.268;
   1:  PR[GP1:91,2] = PR[GP1:90,2] + -37.836;
   1:L PR[91] R[100]mm/sec CNT100;
   1:  PR[GP1:91,1] = PR[GP1:90,1] + 29.427;
   1:  PR[GP1:91,2] = PR[GP1:90,2] + -37.779;
   1:L PR[91] R[100]mm/sec CNT100;
   1:  PR[GP1:91,1] = PR[GP1:90,1] + 30.395;
   1:  PR[GP1:91,2] = PR[GP1:90,2] + -37.570;
   1:L PR[91] R[100]mm/sec CNT100;
   1:  PR[GP1:91,1] = PR[GP1:90,1] + 31.523;
   1:  PR[GP1:91,2] = PR[GP1:90,2] + -37.126;
   1:L PR[91] R[100]mm/sec CNT100;
   1:  PR[GP1:91,1] = PR[GP1:90,1] + 42.568;
   1:  PR[GP1:91,2] = PR[GP1:90,2] + -33.211;
   1:L PR[91] R[100]mm/sec CNT100;
   1:  PR[GP1:91,1] = PR[GP1:90,1] + 43.946;
   1:  PR[GP1:91,2] = PR[GP1:90,2] + -32.357;
   1:L PR[91] R[100]mm/sec CNT100;
   1:  PR[GP1:91,1] = PR[GP1:90,1] + 45.332;
   1:  PR[GP1:91,2] = PR[GP1:90,2] + -31.130;
   1:L PR[91] R[100]mm/sec CNT100;
   1:  PR[GP1:91,1] = PR[GP1:90,1] + 53.286;
   1:  PR[GP1:91,2] = PR[GP1:90,2] + -24.691;
   1:L PR[91] R[100]mm/sec CNT100;
   1:  PR[GP1:91,1] = PR[GP1:90,1] + 54.589;
   1:  PR[GP1:91,2] = PR[GP1:90,2] + -23.000;
   1:L PR[91] R[100]mm/sec CNT100;
   1:  PR[GP1:91,1] = PR[GP1:90,1] + 55.703;
   1:  PR[GP1:91,2] = PR[GP1:90,2] + -20.862;
   1:L PR[91] R[100]mm/sec CNT100;
   1:  PR[GP1:91,1] = PR[GP1:90,1] + 60.360;
   1:  PR[GP1:91,2] = PR[GP1:90,2] + -13.103;
   1:L PR[91] R[100]mm/sec CNT100;
   1:  PR[GP1:91,1] = PR[GP1:90,1] + 61.030;
   1:  PR[GP1:91,2] = PR[GP1:90,2] + -10.860;
   1:L PR[91] R[100]mm/sec CNT100;
   1:  PR[GP1:91,1] = PR[GP1:90,1] + 61.268;
   1:  PR[GP1:91,2] = PR[GP1:90,2] + -8.312;
   1:L PR[91] R[100]mm/sec CNT100;
   1:  PR[GP1:91,1] = PR[GP1:90,1] + 62.791;
   1:  PR[GP1:91,2] = PR[GP1:90,2] + -0.045;
   1:L PR[91] R[100]mm/sec CNT100;
   1:  PR[GP1:91,1] = PR[GP1:90,1] + 62.555;
   1:  PR[GP1:91,2] = PR[GP1:90,2] + 2.506;
   1:L PR[91] R[100]mm/sec CNT100;
   1:  PR[GP1:91,1] = PR[GP1:90,1] + 61.039;
   1:  PR[GP1:91,2] = PR[GP1:90,2] + 10.688;
   1:L PR[91] R[100]mm/sec CNT100;
   1:  PR[GP1:91,1] = PR[GP1:90,1] + 60.355;
   1:  PR[GP1:91,2] = PR[GP1:90,2] + 12.976;
   1:L PR[91] R[100]mm/sec CNT100;
   1:  PR[GP1:91,1] = PR[GP1:90,1] + 59.241;
   1:  PR[GP1:91,2] = PR[GP1:90,2] + 15.135;
   1:L PR[91] R[100]mm/sec CNT100;
   1:  PR[GP1:91,1] = PR[GP1:90,1] + 54.604;
   1:  PR[GP1:91,2] = PR[GP1:90,2] + 22.837;
   1:L PR[91] R[100]mm/sec CNT100;
   1:  PR[GP1:91,1] = PR[GP1:90,1] + 53.281;
   1:  PR[GP1:91,2] = PR[GP1:90,2] + 24.555;
   1:L PR[91] R[100]mm/sec CNT100;
   1:  PR[GP1:91,1] = PR[GP1:90,1] + 51.813;
   1:  PR[GP1:91,2] = PR[GP1:90,2] + 25.867;
   1:L PR[91] R[100]mm/sec CNT100;
   1:  PR[GP1:91,1] = PR[GP1:90,1] + 43.967;
   1:  PR[GP1:91,2] = PR[GP1:90,2] + 32.201;
   1:L PR[91] R[100]mm/sec CNT100;
   1:  PR[GP1:91,1] = PR[GP1:90,1] + 42.567;
   1:  PR[GP1:91,2] = PR[GP1:90,2] + 33.069;
   1:L PR[91] R[100]mm/sec CNT100;
   1:  PR[GP1:91,1] = PR[GP1:90,1] + 41.178;
   1:  PR[GP1:91,2] = PR[GP1:90,2] + 33.624;
   1:L PR[91] R[100]mm/sec CNT100;
   1:  PR[GP1:91,1] = PR[GP1:90,1] + 30.420;
   1:  PR[GP1:91,2] = PR[GP1:90,2] + 37.421;
   1:L PR[91] R[100]mm/sec CNT100;
   1:  PR[GP1:91,1] = PR[GP1:90,1] + 29.432;
   1:  PR[GP1:91,2] = PR[GP1:90,2] + 37.634;
   1:L PR[91] R[100]mm/sec CNT100;
   1:  PR[GP1:91,1] = PR[GP1:90,1] + 28.527;
   1:  PR[GP1:91,2] = PR[GP1:90,2] + 37.668;
   1:L PR[91] R[100]mm/sec CNT100;
   1:  PR[GP1:91,1] = PR[GP1:90,1] + 15.825;
   1:  PR[GP1:91,2] = PR[GP1:90,2] + 37.713;
   1:L PR[91] R[100]mm/sec CNT100;
   1:  PR[GP1:91,1] = PR[GP1:90,1] + 15.476;
   1:  PR[GP1:91,2] = PR[GP1:90,2] + 37.667;
   1:L PR[91] R[100]mm/sec CNT100;
   1:  PR[GP1:91,1] = PR[GP1:90,1] + 5.662;
   1:  PR[GP1:91,2] = PR[GP1:90,2] + 34.275;
   1:L PR[91] R[100]mm/sec CNT100;
   1:  PR[GP1:91,1] = PR[GP1:90,1] + 2.975;
   1:  PR[GP1:91,2] = PR[GP1:90,2] + 33.402;
   1:L PR[91] R[100]mm/sec CNT100;
   1:  PR[GP1:91,2] = PR[GP1:90,2] + 33.399;
   1:L PR[91] R[100]mm/sec CNT100;
   1:  PR[GP1:91,1] = PR[GP1:90,1] + 2.120;
   1:  PR[GP1:91,2] = PR[GP1:90,2] + 32.924;
   1:L PR[91] R[100]mm/sec CNT100;
   1:  ! -- Layer/Ebene 115 -- !;
   1:  PR[91] = PR[90];
   1:  PR[GP1:91,1] = PR[GP1:90,1] + -1.027;
   1:  PR[GP1:91,2] = PR[GP1:90,2] + 33.428;
   1:  PR[GP1:91,3] = PR[GP1:90,3] + 70.455;
   1:L PR[91] R[100]mm/sec CNT100;
   1:  PR[GP1:91,1] = PR[GP1:90,1] + -2.213;
   1:  PR[GP1:91,2] = PR[GP1:90,2] + 33.421;
   1:L PR[91] R[100]mm/sec CNT100;
   1:  PR[GP1:91,1] = PR[GP1:90,1] + -8.618;
   1:  PR[GP1:91,2] = PR[GP1:90,2] + 35.510;
   1:L PR[91] R[100]mm/sec CNT100;
   1:  PR[GP1:91,1] = PR[GP1:90,1] + -15.069;
   1:  PR[GP1:91,2] = PR[GP1:90,2] + 37.740;
   1:L PR[91] R[100]mm/sec CNT100;
   1:  PR[GP1:91,1] = PR[GP1:90,1] + -15.264;
   1:  PR[GP1:91,2] = PR[GP1:90,2] + 37.766;
   1:L PR[91] R[100]mm/sec CNT100;
   1:  PR[GP1:91,1] = PR[GP1:90,1] + -29.050;
   1:  PR[GP1:91,2] = PR[GP1:90,2] + 37.687;
   1:L PR[91] R[100]mm/sec CNT100;
   1:  PR[GP1:91,1] = PR[GP1:90,1] + -29.861;
   1:  PR[GP1:91,2] = PR[GP1:90,2] + 37.512;
   1:L PR[91] R[100]mm/sec CNT100;
   1:  PR[GP1:91,1] = PR[GP1:90,1] + -30.818;
   1:  PR[GP1:91,2] = PR[GP1:90,2] + 37.133;
   1:L PR[91] R[100]mm/sec CNT100;
   1:  PR[GP1:91,1] = PR[GP1:90,1] + -42.189;
   1:  PR[GP1:91,2] = PR[GP1:90,2] + 33.095;
   1:L PR[91] R[100]mm/sec CNT100;
   1:  PR[GP1:91,1] = PR[GP1:90,1] + -43.435;
   1:  PR[GP1:91,2] = PR[GP1:90,2] + 32.319;
   1:L PR[91] R[100]mm/sec CNT100;
   1:  PR[GP1:91,1] = PR[GP1:90,1] + -44.694;
   1:  PR[GP1:91,2] = PR[GP1:90,2] + 31.201;
   1:L PR[91] R[100]mm/sec CNT100;
   1:  PR[GP1:91,1] = PR[GP1:90,1] + -52.921;
   1:  PR[GP1:91,2] = PR[GP1:90,2] + 24.544;
   1:L PR[91] R[100]mm/sec CNT100;
   1:  PR[GP1:91,1] = PR[GP1:90,1] + -54.108;
   1:  PR[GP1:91,2] = PR[GP1:90,2] + 22.999;
   1:L PR[91] R[100]mm/sec CNT100;
   1:  PR[GP1:91,1] = PR[GP1:90,1] + -55.136;
   1:  PR[GP1:91,2] = PR[GP1:90,2] + 21.004;
   1:L PR[91] R[100]mm/sec CNT100;
   1:  PR[GP1:91,1] = PR[GP1:90,1] + -59.970;
   1:  PR[GP1:91,2] = PR[GP1:90,2] + 12.928;
   1:L PR[91] R[100]mm/sec CNT100;
   1:  PR[GP1:91,1] = PR[GP1:90,1] + -60.596;
   1:  PR[GP1:91,2] = PR[GP1:90,2] + 10.807;
   1:L PR[91] R[100]mm/sec CNT100;
   1:  PR[GP1:91,1] = PR[GP1:90,1] + -60.808;
   1:  PR[GP1:91,2] = PR[GP1:90,2] + 8.489;
   1:L PR[91] R[100]mm/sec CNT100;
   1:  PR[GP1:91,1] = PR[GP1:90,1] + -62.391;
   1:  PR[GP1:91,2] = PR[GP1:90,2] + -0.100;
   1:L PR[91] R[100]mm/sec CNT100;
   1:  PR[GP1:91,1] = PR[GP1:90,1] + -62.181;
   1:  PR[GP1:91,2] = PR[GP1:90,2] + -2.423;
   1:L PR[91] R[100]mm/sec CNT100;
   1:  PR[GP1:91,1] = PR[GP1:90,1] + -60.603;
   1:  PR[GP1:91,2] = PR[GP1:90,2] + -10.927;
   1:L PR[91] R[100]mm/sec CNT100;
   1:  PR[GP1:91,1] = PR[GP1:90,1] + -59.964;
   1:  PR[GP1:91,2] = PR[GP1:90,2] + -13.095;
   1:L PR[91] R[100]mm/sec CNT100;
   1:  PR[GP1:91,1] = PR[GP1:90,1] + -58.927;
   1:  PR[GP1:91,2] = PR[GP1:90,2] + -15.127;
   1:L PR[91] R[100]mm/sec CNT100;
   1:  PR[GP1:91,1] = PR[GP1:90,1] + -54.116;
   1:  PR[GP1:91,2] = PR[GP1:90,2] + -23.132;
   1:L PR[91] R[100]mm/sec CNT100;
   1:  PR[GP1:91,1] = PR[GP1:90,1] + -52.907;
   1:  PR[GP1:91,2] = PR[GP1:90,2] + -24.705;
   1:L PR[91] R[100]mm/sec CNT100;
   1:  PR[GP1:91,1] = PR[GP1:90,1] + -51.545;
   1:  PR[GP1:91,2] = PR[GP1:90,2] + -25.927;
   1:L PR[91] R[100]mm/sec CNT100;
   1:  PR[GP1:91,1] = PR[GP1:90,1] + -43.438;
   1:  PR[GP1:91,2] = PR[GP1:90,2] + -32.461;
   1:L PR[91] R[100]mm/sec CNT100;
   1:  PR[GP1:91,1] = PR[GP1:90,1] + -42.170;
   1:  PR[GP1:91,2] = PR[GP1:90,2] + -33.251;
   1:L PR[91] R[100]mm/sec CNT100;
   1:  PR[GP1:91,1] = PR[GP1:90,1] + -40.921;
   1:  PR[GP1:91,2] = PR[GP1:90,2] + -33.753;
   1:L PR[91] R[100]mm/sec CNT100;
   1:  PR[GP1:91,1] = PR[GP1:90,1] + -29.856;
   1:  PR[GP1:91,2] = PR[GP1:90,2] + -37.656;
   1:L PR[91] R[100]mm/sec CNT100;
   1:  PR[GP1:91,1] = PR[GP1:90,1] + -29.025;
   1:  PR[GP1:91,2] = PR[GP1:90,2] + -37.836;
   1:L PR[91] R[100]mm/sec CNT100;
   1:  PR[GP1:91,1] = PR[GP1:90,1] + -28.257;
   1:  PR[GP1:91,2] = PR[GP1:90,2] + -37.865;
   1:L PR[91] R[100]mm/sec CNT100;
   1:  PR[GP1:91,1] = PR[GP1:90,1] + -15.242;
   1:  PR[GP1:91,2] = PR[GP1:90,2] + -37.906;
   1:L PR[91] R[100]mm/sec CNT100;
   1:  PR[GP1:91,1] = PR[GP1:90,1] + -15.040;
   1:  PR[GP1:91,2] = PR[GP1:90,2] + -37.880;
   1:L PR[91] R[100]mm/sec CNT100;
   1:  PR[GP1:91,1] = PR[GP1:90,1] + -14.847;
   1:  PR[GP1:91,2] = PR[GP1:90,2] + -37.819;
   1:L PR[91] R[100]mm/sec CNT100;
   1:  PR[GP1:91,1] = PR[GP1:90,1] + -8.724;
   1:  PR[GP1:91,2] = PR[GP1:90,2] + -35.691;
   1:L PR[91] R[100]mm/sec CNT100;
   1:  PR[GP1:91,1] = PR[GP1:90,1] + -2.213;
   1:  PR[GP1:91,2] = PR[GP1:90,2] + -33.566;
   1:L PR[91] R[100]mm/sec CNT100;
   1:  PR[GP1:91,1] = PR[GP1:90,1] + -0.956;
   1:  PR[GP1:91,2] = PR[GP1:90,2] + -33.572;
   1:L PR[91] R[100]mm/sec CNT100;
   1:  PR[GP1:91,1] = PR[GP1:90,1] + 1.246;
   1:  PR[GP1:91,2] = PR[GP1:90,2] + -33.484;
   1:L PR[91] R[100]mm/sec CNT100;
   1:  PR[GP1:91,1] = PR[GP1:90,1] + 2.180;
   1:  PR[GP1:91,2] = PR[GP1:90,2] + -33.285;
   1:L PR[91] R[100]mm/sec CNT100;
   1:  PR[GP1:91,1] = PR[GP1:90,1] + 2.615;
   1:  PR[GP1:91,2] = PR[GP1:90,2] + -33.635;
   1:L PR[91] R[100]mm/sec CNT100;
   1:  PR[GP1:91,1] = PR[GP1:90,1] + 8.934;
   1:  PR[GP1:91,2] = PR[GP1:90,2] + -35.691;
   1:L PR[91] R[100]mm/sec CNT100;
   1:  PR[GP1:91,1] = PR[GP1:90,1] + 15.257;
   1:  PR[GP1:91,2] = PR[GP1:90,2] + -37.880;
   1:L PR[91] R[100]mm/sec CNT100;
   1:  PR[GP1:91,1] = PR[GP1:90,1] + 15.451;
   1:  PR[GP1:91,2] = PR[GP1:90,2] + -37.905;
   1:L PR[91] R[100]mm/sec CNT100;
   1:  PR[GP1:91,1] = PR[GP1:90,1] + 29.240;
   1:  PR[GP1:91,2] = PR[GP1:90,2] + -37.835;
   1:L PR[91] R[100]mm/sec CNT100;
   1:  PR[GP1:91,1] = PR[GP1:90,1] + 30.050;
   1:  PR[GP1:91,2] = PR[GP1:90,2] + -37.661;
   1:L PR[91] R[100]mm/sec CNT100;
   1:  PR[GP1:91,1] = PR[GP1:90,1] + 31.007;
   1:  PR[GP1:91,2] = PR[GP1:90,2] + -37.284;
   1:L PR[91] R[100]mm/sec CNT100;
   1:  PR[GP1:91,1] = PR[GP1:90,1] + 42.385;
   1:  PR[GP1:91,2] = PR[GP1:90,2] + -33.251;
   1:L PR[91] R[100]mm/sec CNT100;
   1:  PR[GP1:91,1] = PR[GP1:90,1] + 43.623;
   1:  PR[GP1:91,2] = PR[GP1:90,2] + -32.484;
   1:L PR[91] R[100]mm/sec CNT100;
   1:  PR[GP1:91,1] = PR[GP1:90,1] + 44.874;
   1:  PR[GP1:91,2] = PR[GP1:90,2] + -31.376;
   1:L PR[91] R[100]mm/sec CNT100;
   1:  PR[GP1:91,1] = PR[GP1:90,1] + 53.104;
   1:  PR[GP1:91,2] = PR[GP1:90,2] + -24.714;
   1:L PR[91] R[100]mm/sec CNT100;
   1:  PR[GP1:91,1] = PR[GP1:90,1] + 54.305;
   1:  PR[GP1:91,2] = PR[GP1:90,2] + -23.155;
   1:L PR[91] R[100]mm/sec CNT100;
   1:  PR[GP1:91,1] = PR[GP1:90,1] + 55.335;
   1:  PR[GP1:91,2] = PR[GP1:90,2] + -21.178;
   1:L PR[91] R[100]mm/sec CNT100;
   1:  PR[GP1:91,1] = PR[GP1:90,1] + 60.173;
   1:  PR[GP1:91,2] = PR[GP1:90,2] + -13.117;
   1:L PR[91] R[100]mm/sec CNT100;
   1:  PR[GP1:91,1] = PR[GP1:90,1] + 60.798;
   1:  PR[GP1:91,2] = PR[GP1:90,2] + -11.028;
   1:L PR[91] R[100]mm/sec CNT100;
   1:  PR[GP1:91,1] = PR[GP1:90,1] + 61.020;
   1:  PR[GP1:91,2] = PR[GP1:90,2] + -8.647;
   1:L PR[91] R[100]mm/sec CNT100;
   1:  PR[GP1:91,1] = PR[GP1:90,1] + 62.604;
   1:  PR[GP1:91,2] = PR[GP1:90,2] + -0.045;
   1:L PR[91] R[100]mm/sec CNT100;
   1:  PR[GP1:91,1] = PR[GP1:90,1] + 62.384;
   1:  PR[GP1:91,2] = PR[GP1:90,2] + 2.345;
   1:L PR[91] R[100]mm/sec CNT100;
   1:  PR[GP1:91,1] = PR[GP1:90,1] + 60.806;
   1:  PR[GP1:91,2] = PR[GP1:90,2] + 10.855;
   1:L PR[91] R[100]mm/sec CNT100;
   1:  PR[GP1:91,1] = PR[GP1:90,1] + 60.169;
   1:  PR[GP1:91,2] = PR[GP1:90,2] + 12.990;
   1:L PR[91] R[100]mm/sec CNT100;
   1:  PR[GP1:91,1] = PR[GP1:90,1] + 59.129;
   1:  PR[GP1:91,2] = PR[GP1:90,2] + 15.004;
   1:L PR[91] R[100]mm/sec CNT100;
   1:  PR[GP1:91,1] = PR[GP1:90,1] + 54.320;
   1:  PR[GP1:91,2] = PR[GP1:90,2] + 22.992;
   1:L PR[91] R[100]mm/sec CNT100;
   1:  PR[GP1:91,1] = PR[GP1:90,1] + 53.099;
   1:  PR[GP1:91,2] = PR[GP1:90,2] + 24.577;
   1:L PR[91] R[100]mm/sec CNT100;
   1:  PR[GP1:91,1] = PR[GP1:90,1] + 51.744;
   1:  PR[GP1:91,2] = PR[GP1:90,2] + 25.789;
   1:L PR[91] R[100]mm/sec CNT100;
   1:  PR[GP1:91,1] = PR[GP1:90,1] + 43.644;
   1:  PR[GP1:91,2] = PR[GP1:90,2] + 32.328;
   1:L PR[91] R[100]mm/sec CNT100;
   1:  PR[GP1:91,1] = PR[GP1:90,1] + 42.384;
   1:  PR[GP1:91,2] = PR[GP1:90,2] + 33.108;
   1:L PR[91] R[100]mm/sec CNT100;
   1:  PR[GP1:91,1] = PR[GP1:90,1] + 41.133;
   1:  PR[GP1:91,2] = PR[GP1:90,2] + 33.608;
   1:L PR[91] R[100]mm/sec CNT100;
   1:  PR[GP1:91,1] = PR[GP1:90,1] + 30.076;
   1:  PR[GP1:91,2] = PR[GP1:90,2] + 37.512;
   1:L PR[91] R[100]mm/sec CNT100;
   1:  PR[GP1:91,1] = PR[GP1:90,1] + 29.245;
   1:  PR[GP1:91,2] = PR[GP1:90,2] + 37.691;
   1:L PR[91] R[100]mm/sec CNT100;
   1:  PR[GP1:91,1] = PR[GP1:90,1] + 28.481;
   1:  PR[GP1:91,2] = PR[GP1:90,2] + 37.719;
   1:L PR[91] R[100]mm/sec CNT100;
   1:  PR[GP1:91,1] = PR[GP1:90,1] + 15.473;
   1:  PR[GP1:91,2] = PR[GP1:90,2] + 37.765;
   1:L PR[91] R[100]mm/sec CNT100;
   1:  PR[GP1:91,1] = PR[GP1:90,1] + 15.278;
   1:  PR[GP1:91,2] = PR[GP1:90,2] + 37.739;
   1:L PR[91] R[100]mm/sec CNT100;
   1:  PR[GP1:91,1] = PR[GP1:90,1] + 8.829;
   1:  PR[GP1:91,2] = PR[GP1:90,2] + 35.511;
   1:L PR[91] R[100]mm/sec CNT100;
   1:  PR[GP1:91,1] = PR[GP1:90,1] + 2.897;
   1:  PR[GP1:91,2] = PR[GP1:90,2] + 33.583;
   1:L PR[91] R[100]mm/sec CNT100;
   1:  PR[GP1:91,1] = PR[GP1:90,1] + 2.150;
   1:  PR[GP1:91,2] = PR[GP1:90,2] + 33.167;
   1:L PR[91] R[100]mm/sec CNT100;
   1:  ! -- Layer/Ebene 116 -- !;
   1:  PR[91] = PR[90];
   1:  PR[GP1:91,1] = PR[GP1:90,1] + -0.436;
   1:  PR[GP1:91,2] = PR[GP1:90,2] + 33.625;
   1:  PR[GP1:91,3] = PR[GP1:90,3] + 71.065;
   1:L PR[91] R[100]mm/sec CNT100;
   1:  PR[GP1:91,1] = PR[GP1:90,1] + -2.186;
   1:  PR[GP1:91,2] = PR[GP1:90,2] + 33.614;
   1:L PR[91] R[100]mm/sec CNT100;
   1:  PR[GP1:91,1] = PR[GP1:90,1] + -11.784;
   1:  PR[GP1:91,2] = PR[GP1:90,2] + 36.746;
   1:L PR[91] R[100]mm/sec CNT100;
   1:  PR[GP1:91,1] = PR[GP1:90,1] + -14.870;
   1:  PR[GP1:91,2] = PR[GP1:90,2] + 37.813;
   1:L PR[91] R[100]mm/sec CNT100;
   1:  PR[GP1:91,1] = PR[GP1:90,1] + -14.913;
   1:  PR[GP1:91,2] = PR[GP1:90,2] + 37.818;
   1:L PR[91] R[100]mm/sec CNT100;
   1:  PR[GP1:91,1] = PR[GP1:90,1] + -28.862;
   1:  PR[GP1:91,2] = PR[GP1:90,2] + 37.744;
   1:L PR[91] R[100]mm/sec CNT100;
   1:  PR[GP1:91,1] = PR[GP1:90,1] + -29.516;
   1:  PR[GP1:91,2] = PR[GP1:90,2] + 37.603;
   1:L PR[91] R[100]mm/sec CNT100;
   1:  PR[GP1:91,1] = PR[GP1:90,1] + -30.303;
   1:  PR[GP1:91,2] = PR[GP1:90,2] + 37.291;
   1:L PR[91] R[100]mm/sec CNT100;
   1:  PR[GP1:91,1] = PR[GP1:90,1] + -42.006;
   1:  PR[GP1:91,2] = PR[GP1:90,2] + 33.135;
   1:L PR[91] R[100]mm/sec CNT100;
   1:  PR[GP1:91,1] = PR[GP1:90,1] + -43.110;
   1:  PR[GP1:91,2] = PR[GP1:90,2] + 32.447;
   1:L PR[91] R[100]mm/sec CNT100;
   1:  PR[GP1:91,1] = PR[GP1:90,1] + -44.234;
   1:  PR[GP1:91,2] = PR[GP1:90,2] + 31.450;
   1:L PR[91] R[100]mm/sec CNT100;
   1:  PR[GP1:91,1] = PR[GP1:90,1] + -52.737;
   1:  PR[GP1:91,2] = PR[GP1:90,2] + 24.568;
   1:L PR[91] R[100]mm/sec CNT100;
   1:  PR[GP1:91,1] = PR[GP1:90,1] + -53.823;
   1:  PR[GP1:91,2] = PR[GP1:90,2] + 23.155;
